// TwinCAT 3 PLC project SODG11_SSCC610_2403701_PLC
// Title: SSCC6.10
// Company: Sodecia GTAC
// Author: GTAC FW Team
// ProjectVersion: 6.10
// Description: 20250506_release
// libraries:
//   Tc2_Drive, * (Beckhoff Automation GmbH)
//   Tc2_EtherCAT, * (Beckhoff Automation GmbH)
//   Tc2_Math, * (Beckhoff Automation GmbH)
//   Tc2_MC2, * (Beckhoff Automation GmbH)
//   Tc2_MC2_Drive, * (Beckhoff Automation GmbH)
//   Tc2_MDP, * (Beckhoff Automation GmbH)
//   Tc2_Standard, * (Beckhoff Automation GmbH)
//   Tc2_System, * (Beckhoff Automation GmbH)
//   Tc2_TcpIp, * (Beckhoff Automation GmbH)
//   Tc2_Utilities, * (Beckhoff Automation GmbH)
//   Tc3_EventLogger, * (Beckhoff Automation GmbH)
//   Tc3_IPCDiag, * (Beckhoff Automation GmbH)
//   Tc3_Module, * (Beckhoff Automation GmbH)
// project tree:
//   Data types/ATI/ udt_ATI_Input_20150203.TcDUT, udt_ATI_Output_20150203.TcDUT
//   Data types/Beckhoff IO udts/ udt_AdsAddr.TcDUT, udt_AdsAddr_AX5805.TcDUT, udt_CU1128_20180507.TcDUT, udt_ECATMaster_InfoData_20121206.TcDUT, udt_ECATMaster_Status.TcDUT, udt_ECATMaster_Status_20141211.TcDUT, udt_ECATSlave_Status.TcDUT, udt_ECATSlave_StatusADS.TcDUT, udt_ECATSlave_StatusEXT.TcDUT, udt_ECATSlave_Status_CU1128.TcDUT, udt_ECATSlave_Status_EP9128.TcDUT, udt_EK1100.TcDUT, udt_EK1110_20150812.TcDUT, udt_EK1122.TcDUT, udt_EL1004.TcDUT, udt_EL1004_v2.TcDUT, udt_EL1008.TcDUT, udt_EL1904.TcDUT, udt_EL1904_v2.TcDUT, udt_EL2008.TcDUT, udt_EL2008_STAT.TcDUT, udt_EL2008_v2.TcDUT, udt_EL2622.TcDUT, udt_EL2622_STAT.TcDUT, udt_EL2904.TcDUT, udt_EL2904RO.TcDUT, udt_EL2904RO_v2.TcDUT, udt_EL3052.TcDUT, udt_EL6692_20121204.TcDUT, udt_EL6695_20151028.TcDUT, udt_EL6731.TcDUT, udt_EL6900_CMD.TcDUT, udt_EL6900_CMD_20121204.TcDUT, udt_EL6900_DeviceInfoData_20160426.TcDUT, udt_EL6900_SafetyGroup_CMD.TcDUT, udt_EL6900_SafetyGroup_STAT.TcDUT, udt_EL6900_STAT.TcDUT, udt_EL6900_STAT_20160426.TcDUT, udt_EL94xx.TcDUT, udt_EP1008_002.TcDUT, udt_EP1008_002_v2.TcDUT, udt_EP1111.TcDUT, udt_EP1908_002.TcDUT, udt_EP1918.TcDUT, udt_EP1918_CMD_20250213.TcDUT, udt_EP1918_STAT_20250213.TcDUT, udt_EP2028_002.TcDUT, udt_EP2028_002_STAT.TcDUT, udt_EP2028_002_v2.TcDUT, udt_EP2328_0002.TcDUT, udt_EP2624.TcDUT, udt_EP2624_STAT.TcDUT, udt_EP3174_0002.TcDUT, udt_EP6224.TcDUT, udt_EP6224_CMD.TcDUT, udt_EP6224_I.TcDUT, udt_EP9128_20250704.TcDUT, udt_EP9214_CH_CMD_20250704.TcDUT, udt_EP9214_CH_STAT_20250704.TcDUT, udt_EP9214_CMD_20250704.TcDUT, udt_EP9214_DEV_CMD_20250704.TcDUT, udt_EP9214_DEV_STAT_20250704.TcDUT, udt_EP9214_STAT_20250704.TcDUT, udt_EP9224_CH_CMD_20161207.TcDUT, udt_EP9224_CH_STAT_20161207.TcDUT, udt_EP9224_CMD_20161207.TcDUT, udt_EP9224_DEV_CMD_20161207.TcDUT, udt_EP9224_DEV_STAT_20161207.TcDUT, udt_EP9224_STAT_20161207.TcDUT, udt_ProfiMaster_Status.TcDUT, udt_ProfiNet_Status.TcDUT, udt_ProfiNode_Status.TcDUT, udt_SMB_Status_20141211.TcDUT
//   Data types/Discrete Image udts/ udt_ATIxx_Image_20151104.TcDUT, udt_Drive_Image_20160804.TcDUT, udt_Drive_Image_20190816.TcDUT, udt_ECATMaster_Image_20220224.TcDUT, udt_ECATNodeConfig_20200729.TcDUT, udt_ECATNodeData_20221507.TcDUT, udt_ECAT_NodeImage_20200618.TcDUT, udt_EOATxx_Image_20170607.TcDUT, udt_EOATxx_Image_20220715.TcDUT, udt_ESWxx_Image_20150814.TcDUT, udt_FixXX_Input_Image_20180202.TcDUT, udt_FixXX_Output_Image_20220715.TcDUT, udt_FixXX_Output_Image_20250721_CUSTOM.TcDUT, udt_FixXX_Persistent_Input.TcDUT, udt_Fronius_Status_20170531.TcDUT, udt_ICxx_Image.TcDUT, udt_ICxx_Image_20201104.TcDUT, udt_MDxx_Image_20251008.TcDUT, udt_NutWeldLVDT_Input_Image_20250616.TcDUT, udt_NutWeldLVDT_Output_Image_20250616.TcDUT, udt_NWx_Image.TcDUT, udt_ISxx_Image_20241121.TcDUT, udt_PEDxx_Image_20170725.TcDUT, udt_PEDxx_Image_20240808.TcDUT, udt_Reamerxx_Image_20180405.TcDUT, udt_RobotDiscreteNode_Image.TcDUT, udt_RobotDiscreteNode_ImageFSOE_20151028.TcDUT, udt_RobotDiscreteNode_ImageSSCCv46wSAFEOP_20131903.TcDUT, udt_RobotDiscreteNode_ImageSSCCv46_20121204.TcDUT, udt_RobotDiscreteNode_ImageSSCCv46_20131001.TcDUT, udt_SDx_Image.TcDUT, udt_SSxx_Image_20150814.TcDUT, udt_SSxx_Image_20250704.TcDUT, udt_STxx_DiscreteNode_20200212.TcDUT, udt_WaterStand_Image_20220131.TcDUT
//   Data types/Emhart udts/ udt_Emhart_DCE1800_Inputold.TcDUT, udt_Emhart_DCE1800_Outputold.TcDUT, udt_Emhart_TE1500_Input.TcDUT, udt_Emhart_TE1500_Inputa.TcDUT, udt_Emhart_TE1500_Output.TcDUT, udt_Emhart_TE1500_Outputa.TcDUT
//   Data types/FSoE udts/ ST_FSoE_02Byte.TcDUT, ST_FSoE_04Byte.TcDUT, ST_FSoE_06Byte.TcDUT, ST_FSoE_08Byte.TcDUT, ST_FSoE_10Byte.TcDUT, ST_FSoE_12Byte.TcDUT, ST_FSoE_14Byte.TcDUT
//   Data types/Generic udts/ udt_Generic_AdsAddr.TcDUT, udt_Generic_EP9214_20250714.TcDUT, udt_Generic_IC_20150928.TcDUT, udt_Generic_Nok_Data_Grid_20251208.TcDUT, udt_Generic_NutWeldLVDTConfig_20250612.TcDUT, udt_Generic_PD_20220906.TcDUT, udt_Generic_Production_20221007.TcDUT, udt_Generic_ProductReportData_20240909.TcDUT, udt_Generic_Robot_20161202.TcDUT, udt_Generic_Robot_20250711_CUSTOM.TcDUT, udt_Generic_Robot_FBIN_CUSTOM.TcDUT, udt_Generic_Robot_FBIN_20250711_CUSTOM.TcDUT, udt_Generic_Robot_Options_20170531.TcDUT, udt_Generic_Sensor_States_20170801.TcDUT, udt_Generic_ServoDrive_FBIN_20211214.TcDUT, udt_Generic_ShiftCommonConfig_20220420.TcDUT, udt_Generic_ShiftConfigTOD_20160527.TcDUT, udt_Generic_ShiftConfigUDINT_20160531.TcDUT, udt_Generic_ShiftConfig_20160519.TcDUT, udt_IVxx_Input_Image_20250812.TcDUT
//   Data types/Graco udts/ udt_Graco_Input.TcDUT, udt_Graco_Outputs.TcDUT
//   Data types/HardwareDiags/ E_State.TcDUT, udt_HardwareDiags.TcDUT
//   Data types/Keyence/ udt_IV2_DiscreteImage.TcDUT, udt_IV2_Inputs.TcDUT, udt_IV2_Outputs.TcDUT
//   Data types/Robot_udts/ udt_EtherCAT_Kuka_InputBits_20121204.TcDUT, udt_EtherCAT_Kuka_OutputBits_20121204.TcDUT, udt_EtherCAT_Motoman_Input_20151105.TcDUT, udt_EtherCAT_Motoman_Output_20151105.TcDUT, udt_GenericRobot_AnyFieldbus_Input58Bytes.TcDUT, udt_GenericRobot_AnyFieldbus_InputBytes_20220421.TcDUT, udt_GenericRobot_AnyFieldbus_Output58Bytes.TcDUT, udt_GenericRobot_AnyFieldbus_OutputBytes_20220421.TcDUT, udt_GenericRobot_CycleTimes_20170304.TcDUT, udt_Profibus_Motoman_Input.TcDUT, udt_Profibus_Motoman_Input_20121204.TcDUT, udt_Profibus_Motoman_Output.TcDUT, udt_Profibus_Motoman_Output_20121204.TcDUT, udt_SingleAxis_MoveData_20160908.TcDUT, udt_SingleAxis_Position_20150119.TcDUT
//   Data types/Schneider udts/ udt_Schneider_VFD_20180808.TcDUT, udt_Schneider_VFD_Image_20180808.TcDUT, udt_Schneider_VFD_Inputs_20190123.TcDUT, udt_Schneider_VFD_Outputs_20190123.TcDUT
//   Data types/Servo Drive udts/AX5000 Diag/ udt_AX5000Diag.TcDUT
//   Data types/Servo Drive udts/ udt_AX5206_20160804.TcDUT, udt_AX5805_20160804.TcDUT, udt_AX5805_DiagData.TcDUT, udt_EL7211_20150115.TcDUT
//   Data types/SIC/ udt_SIC_Profi_Input_20200727.TcDUT, udt_SIC_Profi_Output_20200727.TcDUT
//   Data types/SmartRay/ udt_PLC_Out_To_SmartRay_IN_20260119.TcDUT, udt_Robot_Out_To_SmartRay_IN_20260119.TcDUT, udt_SmartRay_Out_To_PLC_IN_20260119.TcDUT, udt_SmartRay_Out_To_Robot_IN_20260119.TcDUT
//   Data types/SmartRay/UI udt/ udt_SRxx_DiscreteImage.TcDUT, udt_SRxx_Input_Image.TcDUT, udt_SRxx_ToUI_20260122.TcDUT
//   Data types/SMC udts/ udt_SMC_EX260_Stat.TcDUT, udt_SMC_EX260_ValveBank.TcDUT
//   Data types/Trumpf udts/ udt_EtherCat_Trumpf_InputWords_20171002.TcDUT, udt_EtherCat_Trumpf_OutputWords_20171002.TcDUT, udt_TrumpfImage_20171017.TcDUT
//   Data types/UI udts/GTAC Component IO UI udts/ udt_IVxx_ToUI_20250808.TcDUT, udt_LSRxx_ToUI_20220224.TcDUT, udt_ESWxx_ToUI_20220224.TcDUT, udt_ICxx_ToUI_20220224.TcDUT, udt_MDxx_ToUI_20251008.TcDUT, udt_NWxx_ToUI_20220224.TcDUT, udt_ISxx_ToUI_20241121.TcDUT, udt_ProdReportxx_ToUI_20220224.TcDUT, udt_Rxx_ToUI_20220224.TcDUT, udt_SDxx_ToUI_20220224.TcDUT, udt_SLxx_ToUI_20220224.TcDUT, udt_SSxx_ToUI_20250704.TcDUT, udt_STxx_ToUI_20220224.TcDUT, udt_SDxx_FromUI_20220224.TcDUT, udt_VFDxx_ToUI_20250723.TcDUT
//   Data types/UI udts/ udt_UIcommon_InputPers_20250612.TcDUT, udt_UIcommon_Input_20250616.TcDUT, udt_UIcommon_Output_20251008.TcDUT
//   Global Variables/ Global_Persistent_Variables.TcGVL, Global_Variables.TcGVL, Variable_Configuration.TcGVL
//   POUs/ Faults.TcPOU, GTAC_CONFIG.TcPOU, MAIN.TcPOU, Robot_InterLock_Map.TcPOU
//   POUs/FBs/Diagnose/AX5000 Diag/ FB_AxisDiag_20160810.TcPOU
//   POUs/FBs/ FB_ATI_Changer_20151105.TcPOU, FB_Ax5805_GetInfo_20200609.TcPOU, FB_Clamp_Status.TcPOU, FB_Cylinder_Status.TcPOU, FB_Emhart_20200113.TcPOU, FB_ENET_Com20131205.TcPOU, FB_Graco_Seal_20200716.TcPOU, FB_GTAC_Conveyor_20210303.TcPOU, FB_GTAC_EOAT_20170704.TcPOU, FB_GTAC_ESW_20150814.TcPOU, FB_GTAC_EtherCATMaster_20250723.TcPOU, FB_GTAC_ICxx_20181023.TcPOU, FB_GTAC_IV3_20250730.TcPOU, FB_GTAC_Kuka_CUSTOM.TcPOU, FB_GTAC_Load_Seq_20230302.TcPOU, FB_GTAC_NutWeldLVDT_20250612.TcPOU, FB_GTAC_Motoman_20170531.TcPOU, FB_GTAC_ISxx_20241121.TcPOU, FB_GTAC_Ped_20240808.TcPOU, FB_GTAC_ProcessInterlock_20210526.TcPOU, FB_GTAC_QAcheck_20150529.TcPOU, FB_GTAC_Reamer_20180405.TcPOU, FB_GTAC_MDxx_20251008.TcPOU, FB_GTAC_Reamer_20230328.TcPOU, FB_GTAC_RollDoor_20190108.TcPOU, FB_GTAC_ServoSystem_20211214.TcPOU, FB_GTAC_SS_20250407.TcPOU, FB_GTAC_Valve_20170704.TcPOU, FB_GTAC_WaterStand_20220622.TcPOU, FB_Model_Status.TcPOU, FB_Nok_Datagrid.TcPOU, FB_PP_Sensor.TcPOU, FB_Production_Report_20221007.TcPOU, FB_Pulse_Generator.TcPOU, FB_SCHNEIDERVFD_20180808.TcPOU, FB_SIC_MarkProfi_20200727.TcPOU, FB_SmartRay_20260119.TcPOU, FB_SystemDiags20241206.TcPOU, FB_TripleCylinder_20150625.TcPOU, FB_Trumpf_20180125.TcPOU, FB_UDP_PortCreate20140120.TcPOU, FB_VertiGuard_20260310.TcPOU
//   POUs/Fixtures and EOAT/EOAT/ EOAT04.TcPOU
//   POUs/Fixtures and EOAT/Human/ Fix01.TcPOU, Fix02.TcPOU, Fix03.TcPOU, Fix04.TcPOU, Fix05.TcPOU
//   POUs/Fixtures and EOAT/Internal/ Fix101.TcPOU, Fix102.TcPOU, Fix103.TcPOU, Fix104.TcPOU, Fix105.TcPOU
//   POUs/Fixtures and EOAT/Not_Used/ EOAT01.TcPOU, EOAT02.TcPOU, EOAT03.TcPOU, EOAT05.TcPOU, EOAT06.TcPOU, EOAT07.TcPOU, EOAT08.TcPOU, EOAT09.TcPOU, EOAT10.TcPOU, Fix06.TcPOU, Fix07.TcPOU, Fix08.TcPOU, Fix09.TcPOU, Fix10.TcPOU, Fix106.TcPOU, Fix107.TcPOU, Fix108.TcPOU, Fix109.TcPOU, Fix11.TcPOU, Fix110.TcPOU, Fix111.TcPOU, Fix112.TcPOU, Fix12.TcPOU, Fix13.TcPOU, Fix14.TcPOU, Fix15.TcPOU, Fix16.TcPOU
//   POUs/FUNs/ FUN_GTAC_ASCIItoSTRING.TcPOU, FUN_GTAC_BOOLStoINT.TcPOU, FUN_GTAC_BYTEStoINT.TcPOU, FUN_GTAC_DEGtoINDEX.TcPOU, FUN_GTAC_DINTtoINT.TcPOU, FUN_GTAC_EcatSlaveConnState.TcPOU, FUN_GTAC_EcatSlaveConnState_64bit.TcPOU, FUN_GTAC_FindStringInArray.TcPOU, FUN_GTAC_GenericRobotInputImage_From_KUKAKRC4.TcPOU, FUN_GTAC_GenericRobotInputImage_TO_KUKAKRC4.TcPOU, FUN_GTAC_GenericRobotInputImage_TO_MOTOMAN32.TcPOU, FUN_GTAC_GetNodeFromName.TcPOU, FUN_GTAC_KUKAKRC4_To_GenericRobotOutputImage.TcPOU, FUN_GTAC_MOTOMAN32_TO_GenericRobotOutputImage.TcPOU, FUN_GTAC_NC_Error_Messages.TcPOU, FUN_GTAC_OTSTRUCTtoTOD.TcPOU, FUN_GTAC_OTSTRUCTWrapper.TcPOU, FUN_GTAC_ReturnGrossShiftDuration.TcPOU, FUN_GTAC_ReturnNetShiftDuration.TcPOU, FUN_GTAC_ReturnSetLengthSTR.TcPOU, FUN_GTAC_Scaling.TcPOU, FUN_GTAC_TIMESTRUCTtoTOD.TcPOU, FUN_GTAC_TODtoOTSTRUCT.TcPOU, FUN_GTAC_TODtoUDINT.TcPOU, FUN_GTAC_ZeroSecsInUDINT_Time.TcPOU, FUN_RailMove_To_ICxx.TcPOU
//   POUs/Misc/ Ancillary_Equipment.TcPOU, Cell_Services_Prog.TcPOU, Ped_Stations.TcPOU, Servo_Motion.TcPOU, Task_ID_Record.TcPOU
//   / Standard.TcTTO
// real-time tasks:
//   TASK Standard: cycle T#20ms, priority 11, ADS port 350
// I/O:
//   DEVICE EtherCAT Master (EtherCAT), AmsNetId 172.16.1.120.2.1
//     IC01.T01 (EK1100) [EK1100 EtherCAT Coupler (2A E-Bus)]
//       IC01.T02 (EL6900) [EL6900, TwinSAFE PLC]
//       IC01.T03 (EL1904) [EL1904, 4 Ch. Safety Input 24V, TwinSAFE]
//         modules: Module 1 (FSOES)
//       IC01.T04 (EL1904) [EL1904, 4 Ch. Safety Input 24V, TwinSAFE]
//         modules: Module 1 (FSOES)
//       IC01.T05 (EL1904) [EL1904, 4 Ch. Safety Input 24V, TwinSAFE]
//         modules: Module 1 (FSOES)
//       IC01.T06 (EL1904) [EL1904, 4 Ch. Safety Input 24V, TwinSAFE]
//         modules: Module 1 (FSOES)
//       IC01.T07 (EL1904) [EL1904, 4 Ch. Safety Input 24V, TwinSAFE]
//         modules: Module 1 (FSOES)
//       IC01.T08 (EL1904) [EL1904, 4 Ch. Safety Input 24V, TwinSAFE]
//         modules: Module 1 (FSOES)
//       IC01.T09 (EL2904) [EL2904, 4 Ch. Safety Output 24V, 0.5A, TwinSAFE]
//         modules: Module 1 (FSOES), Module 2 (DO)
//       IC01.T10 (EL2904) [EL2904, 4 Ch. Safety Output 24V, 0.5A, TwinSAFE]
//         modules: Module 1 (FSOES), Module 2 (DO)
//       IC01.T11 (EL9410) [EL9410 E-Bus Power Supplier  (Diagnostics)]
//       IC01.T12 (EL1004) [EL1004 4Ch. Dig. Input 24V, 3ms]
//       IC01.T13 (EL1004) [EL1004 4Ch. Dig. Input 24V, 3ms]
//       IC01.T14 (EL2008) [EL2008 8Ch. Dig. Output 24V, 0.5A]
//       IC01.T15 (EL2622) [EL2622 2Ch. Relay Output, NO (230V AC / 30V DC)]
//       IC01.T16 (EK1122) [EK1122 2 port EtherCAT junction]
//         Fix01.N90 (EP9214-0023) [EP9214-0023 4Ch/4Ch Power Distribution for EtherCAT Box Modules]
//         Fix01.N98  (EP2328-0002) [EP2328-0002 4 CH. Dig. In, 3ms, 4 Ch. Dig. Out 24V, 2A, M12]
//         Fix01.N01 (EP1008-0002) [EP1008-0002 8 Ch. Dig. Input 24V, 3ms, M12]
//         Fix01.N02 (EP1008-0002) [EP1008-0002 8 Ch. Dig. Input 24V, 3ms, M12]
//         Fix01.N03 (EP1008-0002) [EP1008-0002 8 Ch. Dig. Input 24V, 3ms, M12]
//         Fix01.N04 (EP1008-0002) [EP1008-0002 8 Ch. Dig. Input 24V, 3ms, M12]
//         Fix01.N05 (EP1008-0002) [EP1008-0002 8 Ch. Dig. Input 24V, 3ms, M12]
//         Fix01.N06 (EP1008-0002) [EP1008-0002 8 Ch. Dig. Input 24V, 3ms, M12]
//         Fix01.N07 (EP1008-0002) [EP1008-0002 8 Ch. Dig. Input 24V, 3ms, M12]
//         Fix01.N08 (EP1008-0002) [EP1008-0002 8 Ch. Dig. Input 24V, 3ms, M12]
//         Fix01.N09 (EP1008-0002) [EP1008-0002 8 Ch. Dig. Input 24V, 3ms, M12]
//         Fix01.N10 (EP1008-0002) [EP1008-0002 8 Ch. Dig. Input 24V, 3ms, M12]
//         Fix01.N11 (EP1008-0002) [EP1008-0002 8 Ch. Dig. Input 24V, 3ms, M12]
//         Fix01.N12 (EP1008-0002) [EP1008-0002 8 Ch. Dig. Input 24V, 3ms, M12]
//         Fix01.N13 (EP1008-0002) [EP1008-0002 8 Ch. Dig. Input 24V, 3ms, M12]
//         Fix01.N14 (EP1008-0002) [EP1008-0002 8 Ch. Dig. Input 24V, 3ms, M12]
//         Fix01.N15 (EP1008-0002) [EP1008-0002 8 Ch. Dig. Input 24V, 3ms, M12]
//         Fix01.N16 (EP1008-0002) [EP1008-0002 8 Ch. Dig. Input 24V, 3ms, M12]
//         Fix01.N17 (EP1008-0002) [EP1008-0002 8 Ch. Dig. Input 24V, 3ms, M12]
//         Fix01.N18 (EP1008-0002) [EP1008-0002 8 Ch. Dig. Input 24V, 3ms, M12]
//         Fix01.N19 (EP1008-0002) [EP1008-0002 8 Ch. Dig. Input 24V, 3ms, M12]
//         Fix01.N20 (EP1008-0002) [EP1008-0002 8 Ch. Dig. Input 24V, 3ms, M12]
//         Fix01.N21 (EP1008-0002) [EP1008-0002 8 Ch. Dig. Input 24V, 3ms, M12]
//         Fix01.N22 (EP1008-0002) [EP1008-0002 8 Ch. Dig. Input 24V, 3ms, M12]
//         Fix01.N23 (EP1008-0002) [EP1008-0002 8 Ch. Dig. Input 24V, 3ms, M12]
//         Fix01.N24 (EP1008-0002) [EP1008-0002 8 Ch. Dig. Input 24V, 3ms, M12]
//         Fix01.N25 (EP1008-0002) [EP1008-0002 8 Ch. Dig. Input 24V, 3ms, M12]
//         Fix01.N26 (EP1008-0002) [EP1008-0002 8 Ch. Dig. Input 24V, 3ms, M12]
//         Fix01.N27 (EP1008-0002) [EP1008-0002 8 Ch. Dig. Input 24V, 3ms, M12]
//         Fix01.N28 (EP1008-0002) [EP1008-0002 8 Ch. Dig. Input 24V, 3ms, M12]
//         Fix01.N29 (EP1008-0002) [EP1008-0002 8 Ch. Dig. Input 24V, 3ms, M12]
//         Fix01.N30 (EP1008-0002) [EP1008-0002 8 Ch. Dig. Input 24V, 3ms, M12] (disabled)
//         Fix01.N31 (EP1008-0002) [EP1008-0002 8 Ch. Dig. Input 24V, 3ms, M12] (disabled)
//         Fix01.N100 (EX260-SEC1) [EX260-SEC1 EtherCAT SI Unit (32DO_PNP) Rev1.2]
//         Fix01.N101 (EX260-SEC1) [EX260-SEC1 EtherCAT SI Unit (32DO_PNP) Rev1.2]
//         Fix02.N90 (EP9214-0023) [EP9214-0023 4Ch/4Ch Power Distribution for EtherCAT Box Modules]
//         Fix02.N98(EP2328-0002) [EP2328-0002 4 CH. Dig. In, 3ms, 4 Ch. Dig. Out 24V, 2A, M12]
//         Fix02.N01 (EP1008-0002) [EP1008-0002 8 Ch. Dig. Input 24V, 3ms, M12]
//         Fix02.N02 (EP1008-0002) [EP1008-0002 8 Ch. Dig. Input 24V, 3ms, M12]
//         Fix02.N03 (EP1008-0002) [EP1008-0002 8 Ch. Dig. Input 24V, 3ms, M12]
//         Fix02.N04 (EP1008-0002) [EP1008-0002 8 Ch. Dig. Input 24V, 3ms, M12]
//         Fix02.N05 (EP1008-0002) [EP1008-0002 8 Ch. Dig. Input 24V, 3ms, M12]
//         Fix02.N06 (EP1008-0002) [EP1008-0002 8 Ch. Dig. Input 24V, 3ms, M12]
//         Fix02.N07 (EP1008-0002) [EP1008-0002 8 Ch. Dig. Input 24V, 3ms, M12]
//         Fix02.N08 (EP1008-0002) [EP1008-0002 8 Ch. Dig. Input 24V, 3ms, M12]
//         Fix02.N09 (EP1008-0002) [EP1008-0002 8 Ch. Dig. Input 24V, 3ms, M12]
//         Fix02.N10 (EP1008-0002) [EP1008-0002 8 Ch. Dig. Input 24V, 3ms, M12]
//         Fix02.N11 (EP1008-0002) [EP1008-0002 8 Ch. Dig. Input 24V, 3ms, M12]
//         Fix02.N12 (EP1008-0002) [EP1008-0002 8 Ch. Dig. Input 24V, 3ms, M12]
//         Fix02.N13 (EP1008-0002) [EP1008-0002 8 Ch. Dig. Input 24V, 3ms, M12]
//         Fix02.N14 (EP1008-0002) [EP1008-0002 8 Ch. Dig. Input 24V, 3ms, M12]
//         Fix02.N15 (EP1008-0002) [EP1008-0002 8 Ch. Dig. Input 24V, 3ms, M12]
//         Fix02.N16 (EP1008-0002) [EP1008-0002 8 Ch. Dig. Input 24V, 3ms, M12]
//         Fix02.N17 (EP1008-0002) [EP1008-0002 8 Ch. Dig. Input 24V, 3ms, M12]
//         Fix02.N18 (EP1008-0002) [EP1008-0002 8 Ch. Dig. Input 24V, 3ms, M12]
//         Fix02.N19 (EP1008-0002) [EP1008-0002 8 Ch. Dig. Input 24V, 3ms, M12]
//         Fix02.N20 (EP1008-0002) [EP1008-0002 8 Ch. Dig. Input 24V, 3ms, M12]
//         Fix02.N21 (EP1008-0002) [EP1008-0002 8 Ch. Dig. Input 24V, 3ms, M12]
//         Fix02.N22 (EP1008-0002) [EP1008-0002 8 Ch. Dig. Input 24V, 3ms, M12]
//         Fix02.N23 (EP1008-0002) [EP1008-0002 8 Ch. Dig. Input 24V, 3ms, M12]
//         Fix02.N24 (EP1008-0002) [EP1008-0002 8 Ch. Dig. Input 24V, 3ms, M12]
//         Fix02.N25 (EP1008-0002) [EP1008-0002 8 Ch. Dig. Input 24V, 3ms, M12]
//         Fix02.N26 (EP1008-0002) [EP1008-0002 8 Ch. Dig. Input 24V, 3ms, M12]
//         Fix02.N27 (EP1008-0002) [EP1008-0002 8 Ch. Dig. Input 24V, 3ms, M12]
//         Fix02.N28(EP1008-0002) [EP1008-0002 8 Ch. Dig. Input 24V, 3ms, M12]
//         Fix02.N29 (EP1008-0002) [EP1008-0002 8 Ch. Dig. Input 24V, 3ms, M12]
//         Fix02.N30 (EP1008-0002) [EP1008-0002 8 Ch. Dig. Input 24V, 3ms, M12] (disabled)
//         Fix02.N31 (EP1008-0002) [EP1008-0002 8 Ch. Dig. Input 24V, 3ms, M12] (disabled)
//         Fix02.N100 (EX260-SEC1) [EX260-SEC1 EtherCAT SI Unit (32DO_PNP) Rev1.2]
//         Fix02.N101 (EX260-SEC1) [EX260-SEC1 EtherCAT SI Unit (32DO_PNP) Rev1.2]
//       IC01.T17 (EL9011) [EL9011 End Terminal]
//     MD01.N01 (EP1918-0002) [EP1918, 8Ch. Safety Input 24V, TwinSAFE]
//       modules: Module 2 (FSLOGIC)
//     MD01.N02 (EP1008-0002) [EP1008-0002 8 Ch. Dig. Input 24V, 3ms, M12]
//     MD01.N03 (EP2624-0002) [EP2624-0002 4Ch. Relay Output, NO (125V AC / 30V DC)]
//     MD02.N01 (EP1918-0002) [EP1918, 8Ch. Safety Input 24V, TwinSAFE]
//       modules: Module 2 (FSLOGIC)
//     MD02.N02 (EP1008-0002) [EP1008-0002 8 Ch. Dig. Input 24V, 3ms, M12]
//     MD02.N03 (EP2624-0002) [EP2624-0002 4Ch. Relay Output, NO (125V AC / 30V DC)]
//     IC02.T01 (EK1100) [EK1100 EtherCAT Coupler (2A E-Bus)]
//       IC02.T02 (EL6900) [EL6900, TwinSAFE PLC]
//       IC02.T03 (EL1904) [EL1904, 4 Ch. Safety Input 24V, TwinSAFE]
//         modules: Module 1 (FSOES)
//       IC02.T04 (EL1904) [EL1904, 4 Ch. Safety Input 24V, TwinSAFE]
//         modules: Module 1 (FSOES)
//       IC02.T05 (EL1904) [EL1904, 4 Ch. Safety Input 24V, TwinSAFE]
//         modules: Module 1 (FSOES)
//       IC02.T06 (EL1904) [EL1904, 4 Ch. Safety Input 24V, TwinSAFE]
//         modules: Module 1 (FSOES)
//       IC02.T07 (EL1904) [EL1904, 4 Ch. Safety Input 24V, TwinSAFE]
//         modules: Module 1 (FSOES)
//       IC02.T08 (EL1904) [EL1904, 4 Ch. Safety Input 24V, TwinSAFE]
//         modules: Module 1 (FSOES)
//       IC02.T09 (EL2904) [EL2904, 4 Ch. Safety Output 24V, 0.5A, TwinSAFE]
//         modules: Module 1 (FSOES), Module 2 (DO)
//       IC02.T10 (EL2904) [EL2904, 4 Ch. Safety Output 24V, 0.5A, TwinSAFE]
//         modules: Module 1 (FSOES), Module 2 (DO)
//       IC02.T11 (EL9410) [EL9410 E-Bus Power Supplier  (Diagnostics)]
//       IC02.T12 (EL1004) [EL1004 4Ch. Dig. Input 24V, 3ms]
//       IC02.T13 (EL1004) [EL1004 4Ch. Dig. Input 24V, 3ms]
//       IC02.T14 (EL2008) [EL2008 8Ch. Dig. Output 24V, 0.5A]
//       IC02.T15 (EL2622) [EL2622 2Ch. Relay Output, NO (230V AC / 30V DC)]
//       IC02.T16 (EK1122) [EK1122 2 port EtherCAT junction]
//         Fix03.N90 (EP9214-0023) [EP9214-0023 4Ch/4Ch Power Distribution for EtherCAT Box Modules]
//         Fix03.N98  (EP2328-0002) [EP2328-0002 4 CH. Dig. In, 3ms, 4 Ch. Dig. Out 24V, 2A, M12]
//         Fix03.N01 (EP1008-0002) [EP1008-0002 8 Ch. Dig. Input 24V, 3ms, M12]
//         Fix03.N02 (EP1008-0002) [EP1008-0002 8 Ch. Dig. Input 24V, 3ms, M12]
//         Fix03.N03 (EP1008-0002) [EP1008-0002 8 Ch. Dig. Input 24V, 3ms, M12]
//         Fix03.N04 (EP1008-0002) [EP1008-0002 8 Ch. Dig. Input 24V, 3ms, M12]
//         Fix03.N05 (EP1008-0002) [EP1008-0002 8 Ch. Dig. Input 24V, 3ms, M12]
//         Fix03.N06 (EP1008-0002) [EP1008-0002 8 Ch. Dig. Input 24V, 3ms, M12]
//         Fix03.N07 (EP1008-0002) [EP1008-0002 8 Ch. Dig. Input 24V, 3ms, M12]
//         Fix03.N08 (EP1008-0002) [EP1008-0002 8 Ch. Dig. Input 24V, 3ms, M12]
//         Fix03.N09 (EP1008-0002) [EP1008-0002 8 Ch. Dig. Input 24V, 3ms, M12]
//         Fix03.N10 (EP1008-0002) [EP1008-0002 8 Ch. Dig. Input 24V, 3ms, M12]
//         Fix03.N11 (EP1008-0002) [EP1008-0002 8 Ch. Dig. Input 24V, 3ms, M12]
//         Fix03.N12 (EP1008-0002) [EP1008-0002 8 Ch. Dig. Input 24V, 3ms, M12]
//         Fix03.N13 (EP1008-0002) [EP1008-0002 8 Ch. Dig. Input 24V, 3ms, M12]
//         Fix03.N14 (EP1008-0002) [EP1008-0002 8 Ch. Dig. Input 24V, 3ms, M12]
//         Fix03.N15 (EP1008-0002) [EP1008-0002 8 Ch. Dig. Input 24V, 3ms, M12]
//         Fix03.N16 (EP1008-0002) [EP1008-0002 8 Ch. Dig. Input 24V, 3ms, M12]
//         Fix03.N17 (EP1008-0002) [EP1008-0002 8 Ch. Dig. Input 24V, 3ms, M12]
//         Fix03.N18 (EP1008-0002) [EP1008-0002 8 Ch. Dig. Input 24V, 3ms, M12]
//         Fix03.N19 (EP1008-0002) [EP1008-0002 8 Ch. Dig. Input 24V, 3ms, M12]
//         Fix03.N20 (EP1008-0002) [EP1008-0002 8 Ch. Dig. Input 24V, 3ms, M12]
//         Fix03.N21 (EP1008-0002) [EP1008-0002 8 Ch. Dig. Input 24V, 3ms, M12]
//         Fix03.N22 (EP1008-0002) [EP1008-0002 8 Ch. Dig. Input 24V, 3ms, M12]
//         Fix03.N100 (EX260-SEC1) [EX260-SEC1 EtherCAT SI Unit (32DO_PNP) Rev1.2]
//         Fix04.N90 (EP9214-0023) [EP9214-0023 4Ch/4Ch Power Distribution for EtherCAT Box Modules]
//         Fix04.N98  (EP2328-0002) [EP2328-0002 4 CH. Dig. In, 3ms, 4 Ch. Dig. Out 24V, 2A, M12]
//         Fix04.N01 (EP1008-0002) [EP1008-0002 8 Ch. Dig. Input 24V, 3ms, M12]
//         Fix04.N02 (EP1008-0002) [EP1008-0002 8 Ch. Dig. Input 24V, 3ms, M12]
//         Fix04.N03 (EP1008-0002) [EP1008-0002 8 Ch. Dig. Input 24V, 3ms, M12]
//         Fix04.N04 (EP1008-0002) [EP1008-0002 8 Ch. Dig. Input 24V, 3ms, M12]
//         Fix04.N05 (EP1008-0002) [EP1008-0002 8 Ch. Dig. Input 24V, 3ms, M12]
//         Fix04.N06 (EP1008-0002) [EP1008-0002 8 Ch. Dig. Input 24V, 3ms, M12]
//         Fix04.N07 (EP1008-0002) [EP1008-0002 8 Ch. Dig. Input 24V, 3ms, M12]
//         Fix04.N08 (EP1008-0002) [EP1008-0002 8 Ch. Dig. Input 24V, 3ms, M12]
//         Fix04.N09 (EP1008-0002) [EP1008-0002 8 Ch. Dig. Input 24V, 3ms, M12]
//         Fix04.N10 (EP1008-0002) [EP1008-0002 8 Ch. Dig. Input 24V, 3ms, M12]
//         Fix04.N11 (EP1008-0002) [EP1008-0002 8 Ch. Dig. Input 24V, 3ms, M12]
//         Fix04.N12 (EP1008-0002) [EP1008-0002 8 Ch. Dig. Input 24V, 3ms, M12]
//         Fix04.N13 (EP1008-0002) [EP1008-0002 8 Ch. Dig. Input 24V, 3ms, M12]
//         Fix04.N14 (EP1008-0002) [EP1008-0002 8 Ch. Dig. Input 24V, 3ms, M12]
//         Fix04.N15 (EP1008-0002) [EP1008-0002 8 Ch. Dig. Input 24V, 3ms, M12]
//         Fix04.N16 (EP1008-0002) [EP1008-0002 8 Ch. Dig. Input 24V, 3ms, M12]
//         Fix04.N17 (EP1008-0002) [EP1008-0002 8 Ch. Dig. Input 24V, 3ms, M12]
//         Fix04.N18 (EP1008-0002) [EP1008-0002 8 Ch. Dig. Input 24V, 3ms, M12]
//         Fix04.N19 (EP1008-0002) [EP1008-0002 8 Ch. Dig. Input 24V, 3ms, M12]
//         Fix04.N20 (EP1008-0002) [EP1008-0002 8 Ch. Dig. Input 24V, 3ms, M12]
//         Fix04.N21 (EP1008-0002) [EP1008-0002 8 Ch. Dig. Input 24V, 3ms, M12]
//         Fix04.N22 (EP1008-0002) [EP1008-0002 8 Ch. Dig. Input 24V, 3ms, M12] (disabled)
//         Fix04.N100 (EX260-SEC1) [EX260-SEC1 EtherCAT SI Unit (32DO_PNP) Rev1.2]
//       IC02.T17 (EL9011) [EL9011 End Terminal]
//     ESW03.N01 (EP1908) [EP1908, 8 Ch. Safety Input 24V, TwinSAFE]
//       modules: Module 1 (FSOE)
//     R5.T01 (EK1100) [EK1100 EtherCAT Coupler (2A E-Bus)]
//       R5.T02 (EL6900) [EL6900, TwinSAFE PLC]
//       R5.T03 (EL1904) [EL1904, 4 Ch. Safety Input 24V, TwinSAFE]
//         modules: Module 1 (FSOES)
//       R5.T04 (EK1122) [EK1122 2 port EtherCAT junction]
//         R5.Reamer[1].N01 (EP1008-0002) [EP1008-0002 8 Ch. Dig. Input 24V, 3ms, M12]
//         R5.Reamer[1].N30 (EP2028-0002) [EP2028-0002 8 Ch. Dig. Output 24V, 2A, M12]
//     R5.RT02 (EL6695-1001) [KRC4 secondary EL6695-1001]
//       modules: Module 1 (Sync Inputs), Module 2 (Safety Data (8 Byte)), Module 3 (Default IO)
//     R6.T01 (EK1100) [EK1100 EtherCAT Coupler (2A E-Bus)]
//       R6.T02 (EL6900) [EL6900, TwinSAFE PLC]
//       R6.T03 (EL1904) [EL1904, 4 Ch. Safety Input 24V, TwinSAFE]
//         modules: Module 1 (FSOES)
//       R6.T04 (EK1122) [EK1122 2 port EtherCAT junction]
//         R6.Reamer[1].N01 (EP1008-0002) [EP1008-0002 8 Ch. Dig. Input 24V, 3ms, M12]
//         R6.Reamer[1].N30 (EP2028-0002) [EP2028-0002 8 Ch. Dig. Output 24V, 2A, M12]
//     R6.RT02 (EL6695-1001) [KRC4 secondary EL6695-1001]
//       modules: Module 1 (Sync Inputs), Module 2 (Safety Data (8 Byte)), Module 3 (Default IO)
//     R10.T01 (EK1100) [EK1100 EtherCAT Coupler (2A E-Bus)]
//       R10.T02 (EL6900) [EL6900, TwinSAFE PLC]
//       R10.T03 (EL1904) [EL1904, 4 Ch. Safety Input 24V, TwinSAFE]
//         modules: Module 1 (FSOES)
//       R10.T04 (EK1122) [EK1122 2 port EtherCAT junction]
//     R10.RT02 (EL6695-1001) [KRC4 secondary EL6695-1001]
//       modules: Module 1 (Sync Inputs), Module 2 (Safety Data (8 Byte)), Module 3 (Default IO)
//     R11.T01 (EK1100) [EK1100 EtherCAT Coupler (2A E-Bus)]
//       R11.T02 (EL6900) [EL6900, TwinSAFE PLC]
//       R11.T03 (EL1904) [EL1904, 4 Ch. Safety Input 24V, TwinSAFE]
//         modules: Module 1 (FSOES)
//       R11.T04 (EK1122) [EK1122 2 port EtherCAT junction]
//     R11.RT02 (EL6695-1001) [KRC4 secondary EL6695-1001]
//       modules: Module 1 (Sync Inputs), Module 2 (Safety Data (8 Byte)), Module 3 (Default IO)
//     IC03.T01 (EK1100) [EK1100 EtherCAT Coupler (2A E-Bus)]
//       IC03.T02 (EL6900) [EL6900, TwinSAFE PLC]
//       IC03.T03 (EL1904) [EL1904, 4 Ch. Safety Input 24V, TwinSAFE]
//         modules: Module 1 (FSOES)
//       IC03.T04 (EL1904) [EL1904, 4 Ch. Safety Input 24V, TwinSAFE]
//         modules: Module 1 (FSOES)
//       IC03.T05 (EL1904) [EL1904, 4 Ch. Safety Input 24V, TwinSAFE]
//         modules: Module 1 (FSOES)
//       IC03.T06 (EL1904) [EL1904, 4 Ch. Safety Input 24V, TwinSAFE]
//         modules: Module 1 (FSOES)
//       IC03.T07 (EL1904) [EL1904, 4 Ch. Safety Input 24V, TwinSAFE]
//         modules: Module 1 (FSOES)
//       IC03.T08 (EL1904) [EL1904, 4 Ch. Safety Input 24V, TwinSAFE]
//         modules: Module 1 (FSOES)
//       IC03.T09 (EL2904) [EL2904, 4 Ch. Safety Output 24V, 0.5A, TwinSAFE]
//         modules: Module 1 (FSOES), Module 2 (DO)
//       IC03.T10 (EL2904) [EL2904, 4 Ch. Safety Output 24V, 0.5A, TwinSAFE]
//         modules: Module 1 (FSOES), Module 2 (DO)
//       IC03.T11 (EL9410) [EL9410 E-Bus Power Supplier  (Diagnostics)]
//       IC03.T12 (EL1004) [EL1004 4Ch. Dig. Input 24V, 3ms]
//       IC03.T13 (EL1004) [EL1004 4Ch. Dig. Input 24V, 3ms]
//       IC03.T14 (EL2008) [EL2008 8Ch. Dig. Output 24V, 0.5A]
//       IC03.T15 (EL2622) [EL2622 2Ch. Relay Output, NO (230V AC / 30V DC)]
//       IC03.T16 (EK1122) [EK1122 2 port EtherCAT junction]
//         Fix05.N01 (EP1008-0002) [EP1008-0002 8 Ch. Dig. Input 24V, 3ms, M12]
//         Fix05.N02 (EP1008-0002) [EP1008-0002 8 Ch. Dig. Input 24V, 3ms, M12]
//         Fix05.N03 (EP1008-0002) [EP1008-0002 8 Ch. Dig. Input 24V, 3ms, M12]
//         Fix05.N04 (EP1008-0002) [EP1008-0002 8 Ch. Dig. Input 24V, 3ms, M12]
//         Fix05.N100 (EX260-SEC1) [EX260-SEC1 EtherCAT SI Unit (32DO_PNP) Rev1.2]
//         Fix102.N01 (EP1008-0002) [EP1008-0002 8 Ch. Dig. Input 24V, 3ms, M12]
//         Fix102.N02 (EP1008-0002) [EP1008-0002 8 Ch. Dig. Input 24V, 3ms, M12]
//         Fix102.N03 (EP1008-0002) [EP1008-0002 8 Ch. Dig. Input 24V, 3ms, M12]
//         Fix102.N04 (EP1008-0002) [EP1008-0002 8 Ch. Dig. Input 24V, 3ms, M12]
//         Fix102.N100 (EX260-SEC1) [EX260-SEC1 EtherCAT SI Unit (32DO_PNP) Rev1.2]
//         QA_Fix102CAM1 (DL-EC1A) [DL-EC1A] (disabled)
//         QA_Fix102CAM2 (DL-EC1A)
//       IC03.T17 (EL9011) [EL9011 End Terminal]
//     ESW02.N01 (EP1908) [EP1908, 8 Ch. Safety Input 24V, TwinSAFE]
//       modules: Module 1 (FSOE)
//     IS01.T01 (EK1100) [EK1100 EtherCAT Coupler (2A E-Bus)]
//       IS01.T02 (EL6900) [EL6900, TwinSAFE PLC]
//       IS01.T03 (EL1904) [EL1904, 4 Ch. Safety Input 24V, TwinSAFE]
//         modules: Module 1 (FSOES)
//       IS01.T04 (EL2904) [EL2904, 4 Ch. Safety Output 24V, 0.5A, TwinSAFE]
//         modules: Module 1 (FSOES), Module 2 (DO)
//       IS01.T05 (EL6731) [EL6731 PROFIBUS DP Master]
//       IS01.T06 (EK1110) [EK1110 EtherCAT extension]
//     SS01.N01 (EP9128-0021) [EP9128-0021 8x EtherCAT junction]
//       Fix101.N01 (EP1008-0002) [EP1008-0002 8 Ch. Dig. Input 24V, 3ms, M12]
//       Fix101.N02 (EP1008-0002) [EP1008-0002 8 Ch. Dig. Input 24V, 3ms, M12]
//       Fix101.N03 (EP1008-0002) [EP1008-0002 8 Ch. Dig. Input 24V, 3ms, M12]
//       Fix101.N04 (EP1008-0002) [EP1008-0002 8 Ch. Dig. Input 24V, 3ms, M12]
//       Fix101.N100 (EX260-SEC1) [EX260-SEC1 EtherCAT SI Unit (32DO_PNP) Rev1.2]
//       VertiGuard.N01 (EP2028-0002) [EP2028-0002 8 Ch. Dig. Output 24V, 2A, M12]
//       VertiGuard.N02 (EP1908) [EP1908, 8 Ch. Safety Input 24V, TwinSAFE ]
//         modules: Module 1 (FSOE)
//       Term 299 (EP9128-1021) [EP9128-1021 8x EtherCAT junction - Dev A]
//         Fix103.N01 (EP1008-0002) [EP1008-0002 8 Ch. Dig. Input 24V, 3ms, M12] (disabled)
//         Fix103.N02 (EP1008-0002) [EP1008-0002 8 Ch. Dig. Input 24V, 3ms, M12] (disabled)
//         VFD01 (ATV320 EtherCAT) [ATV320 EtherCAT] (disabled)
//         Fix104.N01 (EP1008-0002) [EP1008-0002 8 Ch. Dig. Input 24V, 3ms, M12] (disabled)
//         Fix104.N02 (EP1008-0002) [EP1008-0002 8 Ch. Dig. Input 24V, 3ms, M12] (disabled)
//         VFD02 (ATV320 EtherCAT) [ATV320 EtherCAT] (disabled)
//         Fix105.N01 (EP1008-0002)
//         Fix105.N02 (EP1008-0002)
//       Term 301 (EP9128-2021) [EP9128-2021 8x EtherCAT junction - Dev B]
//     SS01.N02 (EP1008-0002) [EP1008-0002 8 Ch. Dig. Input 24V, 3ms, M12]
//     SS01.N03 (EP2028-0002) [EP2028-0002 8 Ch. Dig. Output 24V, 2A, M12]
//     SS01.N04 (EP9214-0023) [EP9214-0023 4Ch/4Ch Power Distribution for EtherCAT Box Modules]
//     R4.T01 (EK1100) [EK1100 EtherCAT Coupler (2A E-Bus)]
//       R4.T02 (EL6900) [EL6900, TwinSAFE PLC]
//       R4.T03 (EL1904) [EL1904, 4 Ch. Safety Input 24V, TwinSAFE]
//         modules: Module 1 (FSOES)
//       R4.T04 (EK1122) [EK1122 2 port EtherCAT junction]
//         EOAT04.N00 (EP1111-0002) [EP1111-0000 ID-Switch]
//         EOAT04.N01 (EP1008-0002) [EP1008-0002 8 Ch. Dig. Input 24V, 3ms, M12]
//         EOAT04.N02 (EP1008-0002) [EP1008-0002 8 Ch. Dig. Input 24V, 3ms, M12]
//         EOAT04.N03 (EP1008-0002) [EP1008-0002 8 Ch. Dig. Input 24V, 3ms, M12]
//         EOAT04.N04 (EP1008-0002) [EP1008-0002 8 Ch. Dig. Input 24V, 3ms, M12]
//         EOAT04.N100 (EX260-SEC1) [EX260-SEC1 EtherCAT SI Unit (32DO_PNP) Rev1.2]
//     R4.RT02 (EL6695-1001) [KRC4 secondary EL6695-1001]
//       modules: Module 1 (Sync Inputs), Module 2 (Safety Data (8 Byte)), Module 3 (Default IO)
//     R1.T01 (EK1100) [EK1100 EtherCAT Coupler (2A E-Bus)]
//       R1.T02 (EL6900) [EL6900, TwinSAFE PLC]
//       R1.T03 (EL1904) [EL1904, 4 Ch. Safety Input 24V, TwinSAFE]
//         modules: Module 1 (FSOES)
//       R1.T04 (EK1122) [EK1122 2 port EtherCAT junction]
//         R1.Reamer[1].N01 (EP1008-0002) [EP1008-0002 8 Ch. Dig. Input 24V, 3ms, M12]
//         R1.Reamer[1].N30 (EP2028-0002) [EP2028-0002 8 Ch. Dig. Output 24V, 2A, M12]
//     R1.RT02 (EL6695-1001) [KRC4 secondary EL6695-1001]
//       modules: Module 1 (Sync Inputs), Module 2 (Safety Data (8 Byte)), Module 3 (Default IO)
//     R2.T01 (EK1100) [EK1100 EtherCAT Coupler (2A E-Bus)]
//       R2.T02 (EL6900) [EL6900, TwinSAFE PLC]
//       R2.T03 (EL1904) [EL1904, 4 Ch. Safety Input 24V, TwinSAFE]
//         modules: Module 1 (FSOES)
//       R2.T04 (EK1122) [EK1122 2 port EtherCAT junction]
//         R2.Reamer[1].N01 (EP1008-0002) [EP1008-0002 8 Ch. Dig. Input 24V, 3ms, M12]
//         R2.Reamer[1].N30 (EP2028-0002) [EP2028-0002 8 Ch. Dig. Output 24V, 2A, M12]
//     R2.RT02 (EL6695-1001) [KRC4 secondary EL6695-1001]
//       modules: Module 1 (Sync Inputs), Module 2 (Safety Data (8 Byte)), Module 3 (Default IO)
//     R3.T01 (EK1100) [EK1100 EtherCAT Coupler (2A E-Bus)]
//       R3.T02 (EL6900) [EL6900, TwinSAFE PLC]
//       R3.T03 (EL1904) [EL1904, 4 Ch. Safety Input 24V, TwinSAFE]
//         modules: Module 1 (FSOES)
//       R3.T04 (EK1122) [EK1122 2 port EtherCAT junction]
//         R3.Reamer[1].N01 (EP1008-0002) [EP1008-0002 8 Ch. Dig. Input 24V, 3ms, M12]
//         R3.Reamer[1].N30 (EP2028-0002) [EP2028-0002 8 Ch. Dig. Output 24V, 2A, M12]
//     R3.RT02 (EL6695-1001) [KRC4 secondary EL6695-1001]
//       modules: Module 1 (Sync Inputs), Module 2 (Safety Data (8 Byte)), Module 3 (Default IO)
//     ESW01.N01 (EP1908) [EP1908, 8 Ch. Safety Input 24V, TwinSAFE]
//       modules: Module 1 (FSOE)
//     R8.T01 (EK1100) [EK1100 EtherCAT Coupler (2A E-Bus)]
//       R8.T02 (EL6900) [EL6900, TwinSAFE PLC]
//       R8.T03 (EL1904) [EL1904, 4 Ch. Safety Input 24V, TwinSAFE]
//         modules: Module 1 (FSOES)
//       R8.T04 (EK1122) [EK1122 2 port EtherCAT junction]
//         R8.Reamer[1].N01 (EP1008-0002) [EP1008-0002 8 Ch. Dig. Input 24V, 3ms, M12]
//         R8.Reamer[1].N30 (EP2028-0002) [EP2028-0002 8 Ch. Dig. Output 24V, 2A, M12]
//     R8.RT02 (EL6695-1001) [KRC4 secondary EL6695-1001]
//       modules: Module 1 (Sync Inputs), Module 2 (Safety Data (8 Byte)), Module 3 (Default IO)
//     R9.T01 (EK1100) [EK1100 EtherCAT Coupler (2A E-Bus)]
//       R9.T02 (EL6900) [EL6900, TwinSAFE PLC]
//       R9.T03 (EL1904) [EL1904, 4 Ch. Safety Input 24V, TwinSAFE]
//         modules: Module 1 (FSOES)
//       R9.T04 (EK1122) [EK1122 2 port EtherCAT junction]
//         R9.Reamer[1].N01 (EP1008-0002) [EP1008-0002 8 Ch. Dig. Input 24V, 3ms, M12]
//         R9.Reamer[1].N30 (EP2028-0002) [EP2028-0002 8 Ch. Dig. Output 24V, 2A, M12]
//     R9.RT02 (EL6695-1001) [KRC4 secondary EL6695-1001]
//       modules: Module 1 (Sync Inputs), Module 2 (Safety Data (8 Byte)), Module 3 (Default IO)
//     R7.T01 (EK1100) [EK1100 EtherCAT Coupler (2A E-Bus)]
//       R7.T02 (EL6900) [EL6900, TwinSAFE PLC]
//       R7.T03 (EL1904) [EL1904, 4 Ch. Safety Input 24V, TwinSAFE]
//         modules: Module 1 (FSOES)
//       R7.T04 (EK1122) [EK1122 2 port EtherCAT junction]
//         R7.Reamer[1].N01 (EP1008-0002) [EP1008-0002 8 Ch. Dig. Input 24V, 3ms, M12]
//         R7.Reamer[1].N30 (EP2028-0002) [EP2028-0002 8 Ch. Dig. Output 24V, 2A, M12]
//     R7.RT02 (EL6695-1001) [KRC4 secondary EL6695-1001]
//       modules: Module 1 (Sync Inputs), Module 2 (Safety Data (8 Byte)), Module 3 (Default IO)
//     Fix01.N32_42 (EP1111-0000) [EP1111-0000 ID-Switch]
//     Fix01.N33_42 (EP1008-0002) [EP1008-0002 8 Ch. Dig. Input 24V, 3ms, M12]
//     Fix01.N34_43 (EP1111-0000) [EP1111-0000 ID-Switch]
//     Fix01.N35_43 (EP1008-0002) [EP1008-0002 8 Ch. Dig. Input 24V, 3ms, M12]
//     Fix01.N36_44 (EP1111-0000) [EP1111-0000 ID-Switch]
//     Fix01.N37_44 (EP1008-0002) [EP1008-0002 8 Ch. Dig. Input 24V, 3ms, M12]
//     Fix01.N38_45 (EP1111-0000) [EP1111-0000 ID-Switch]
//     Fix01.N39_45 (EP1008-0002) [EP1008-0002 8 Ch. Dig. Input 24V, 3ms, M12]
//     Fix01.N40_46 (EP1111-0000) [EP1111-0000 ID-Switch]
//     Fix01.N41_46 (EP1008-0002) [EP1008-0002 8 Ch. Dig. Input 24V, 3ms, M12]
//     Fix01.N42_47 (EP1111-0000) [EP1111-0000 ID-Switch]
//     Fix01.N43_47 (EP1008-0002) [EP1008-0002 8 Ch. Dig. Input 24V, 3ms, M12]
//     Fix02.N32_42 (EP1111-0000) [EP1111-0000 ID-Switch]
//     Fix02.N33_42 (EP1008-0002) [EP1008-0002 8 Ch. Dig. Input 24V, 3ms, M12]
//     Fix02.N34_43 (EP1111-0000) [EP1111-0000 ID-Switch]
//     Fix02.N35_43 (EP1008-0002) [EP1008-0002 8 Ch. Dig. Input 24V, 3ms, M12]
//     Fix02.N36_44 (EP1111-0000) [EP1111-0000 ID-Switch]
//     Fix02.N37_44 (EP1008-0002) [EP1008-0002 8 Ch. Dig. Input 24V, 3ms, M12]
//     Fix02.N38_45 (EP1111-0000) [EP1111-0000 ID-Switch]
//     Fix02.N39_45 (EP1008-0002) [EP1008-0002 8 Ch. Dig. Input 24V, 3ms, M12]
//     Fix02.N40_46 (EP1111-0000) [EP1111-0000 ID-Switch]
//     Fix02.N41_46 (EP1008-0002) [EP1008-0002 8 Ch. Dig. Input 24V, 3ms, M12]
//     Fix02.N42_47 (EP1111-0000) [EP1111-0000 ID-Switch]
//     Fix02.N43_47 (EP1008-0002) [EP1008-0002 8 Ch. Dig. Input 24V, 3ms, M12]
//   DEVICE PD01.T05 (EL6731) (disabled), AmsNetId 172.16.1.191.8.1
//     SIC01.N10 (GSD Box) (UNIGATE IC - Profibus) // Vendor: Deutschmann Automation GmbH Revision: V1.4
//     SIC01.N20 (GSD Box) (UNIGATE IC - Profibus) // Vendor: Deutschmann Automation GmbH Revision: V1.4
// variable links:
//   EtherCAT Master (EtherCAT) <-> EtherCAT Master (EtherCAT)/ESW01.N01 (EP1908)
//     IC01.T01 (EK1100)/IC01.T02 (EL6900)/ConnectionInputs/Message_9 TxPDO <-> Module 1 (FSOE)/FSOE Outputs/FSOE
//     IC01.T01 (EK1100)/IC01.T02 (EL6900)/ConnectionOutputs/Message_9 RxPDO <-> Module 1 (FSOE)/FSOE Inputs/FSOE
//   EtherCAT Master (EtherCAT) <-> EtherCAT Master (EtherCAT)/ESW02.N01 (EP1908)
//     IC01.T01 (EK1100)/IC01.T02 (EL6900)/ConnectionInputs/Message_10 TxPDO <-> Module 1 (FSOE)/FSOE Outputs/FSOE
//   EtherCAT Master (EtherCAT) <-> EtherCAT Master (EtherCAT)/ESW03.N01 (EP1908)
//     IC01.T01 (EK1100)/IC01.T02 (EL6900)/ConnectionOutputs/Message_11 RxPDO <-> Module 1 (FSOE)/FSOE Inputs/FSOE
//   EtherCAT Master (EtherCAT) <-> EtherCAT Master (EtherCAT)/IC01.T01 (EK1100)/IC01.T02 (EL6900)
//     ESW02.N01 (EP1908)/Module 1 (FSOE)/FSOE Inputs/FSOE <-> ConnectionOutputs/Message_10 RxPDO
//     ESW03.N01 (EP1908)/Module 1 (FSOE)/FSOE Outputs/FSOE <-> ConnectionInputs/Message_11 TxPDO
//     IC01.T01 (EK1100)/IC01.T03 (EL1904)/Module 1 (FSOES)/RxPDO/FSOE <-> ConnectionInputs/Message_1 TxPDO
//     IC01.T01 (EK1100)/IC01.T05 (EL1904)/Module 1 (FSOES)/RxPDO/FSOE <-> ConnectionInputs/Message_5 TxPDO
//     IC01.T01 (EK1100)/IC01.T07 (EL1904)/Module 1 (FSOES)/RxPDO/FSOE <-> ConnectionInputs/Message_6 TxPDO
//     IC01.T01 (EK1100)/IC01.T08 (EL1904)/Module 1 (FSOES)/RxPDO/FSOE <-> ConnectionInputs/Message_3 TxPDO
//     IC01.T01 (EK1100)/IC01.T09 (EL2904)/Module 1 (FSOES)/RxPDO/FSOE <-> ConnectionInputs/Message_7 TxPDO
//     IC01.T01 (EK1100)/IC01.T10 (EL2904)/Module 1 (FSOES)/RxPDO/FSOE <-> ConnectionInputs/Message_8 TxPDO
//     IC01.T01 (EK1100)/IC01.T03 (EL1904)/Module 1 (FSOES)/TxPDO/FSOE <-> ConnectionOutputs/Message_1 RxPDO
//     IC01.T01 (EK1100)/IC01.T04 (EL1904)/Module 1 (FSOES)/TxPDO/FSOE <-> ConnectionOutputs/Message_4 RxPDO
//     IC01.T01 (EK1100)/IC01.T06 (EL1904)/Module 1 (FSOES)/TxPDO/FSOE <-> ConnectionOutputs/Message_2 RxPDO
//     IC01.T01 (EK1100)/IC01.T07 (EL1904)/Module 1 (FSOES)/TxPDO/FSOE <-> ConnectionOutputs/Message_6 RxPDO
//     IC01.T01 (EK1100)/IC01.T10 (EL2904)/Module 1 (FSOES)/TxPDO/FSOE <-> ConnectionOutputs/Message_8 RxPDO
//     IC02.T01 (EK1100)/IC02.T02 (EL6900)/ConnectionInputs/Message_9 TxPDO <-> ConnectionOutputs/Message_12 RxPDO
//     IC02.T01 (EK1100)/IC02.T02 (EL6900)/ConnectionOutputs/Message_9 RxPDO <-> ConnectionInputs/Message_12 TxPDO
//     IS01.T01 (EK1100)/IS01.T02 (EL6900)/ConnectionInputs/Message_3 TxPDO <-> ConnectionOutputs/Message_43 RxPDO
//     MD01.N01 (EP1918-0002)/ConnectionOutputs/Message_8 RxPDO <-> ConnectionInputs/Message_105 TxPDO
//     MD02.N01 (EP1918-0002)/ConnectionOutputs/Message_8 RxPDO <-> ConnectionInputs/Message_106 TxPDO
//     MD02.N01 (EP1918-0002)/ConnectionInputs/Message_8 TxPDO <-> ConnectionOutputs/Message_106 RxPDO
//     R10.T01 (EK1100)/R10.T02 (EL6900)/ConnectionInputs/Message_2 TxPDO <-> ConnectionOutputs/Message_27 RxPDO
//     R2.T01 (EK1100)/R2.T02 (EL6900)/ConnectionInputs/Message_2 TxPDO <-> ConnectionOutputs/Message_19 RxPDO
//     R3.T01 (EK1100)/R3.T02 (EL6900)/ConnectionInputs/Message_2 TxPDO <-> ConnectionOutputs/Message_20 RxPDO
//     R4.T01 (EK1100)/R4.T02 (EL6900)/ConnectionInputs/Message_2 TxPDO <-> ConnectionOutputs/Message_21 RxPDO
//     R7.T01 (EK1100)/R7.T02 (EL6900)/ConnectionInputs/Message_2 TxPDO <-> ConnectionOutputs/Message_24 RxPDO
//     R9.T01 (EK1100)/R9.T02 (EL6900)/ConnectionInputs/Message_2 TxPDO <-> ConnectionOutputs/Message_26 RxPDO
//     R3.T01 (EK1100)/R3.T02 (EL6900)/ConnectionOutputs/Message_2 RxPDO <-> ConnectionInputs/Message_20 TxPDO
//     R5.T01 (EK1100)/R5.T02 (EL6900)/ConnectionOutputs/Message_2 RxPDO <-> ConnectionInputs/Message_22 TxPDO
//     R7.T01 (EK1100)/R7.T02 (EL6900)/ConnectionOutputs/Message_2 RxPDO <-> ConnectionInputs/Message_24 TxPDO
//     R8.T01 (EK1100)/R8.T02 (EL6900)/ConnectionOutputs/Message_2 RxPDO <-> ConnectionInputs/Message_25 TxPDO
//   EtherCAT Master (EtherCAT) <-> EtherCAT Master (EtherCAT)/IC01.T01 (EK1100)/IC01.T04 (EL1904)
//     IC01.T01 (EK1100)/IC01.T02 (EL6900)/ConnectionInputs/Message_4 TxPDO <-> Module 1 (FSOES)/RxPDO/FSOE
//   EtherCAT Master (EtherCAT) <-> EtherCAT Master (EtherCAT)/IC01.T01 (EK1100)/IC01.T05 (EL1904)
//     IC01.T01 (EK1100)/IC01.T02 (EL6900)/ConnectionOutputs/Message_5 RxPDO <-> Module 1 (FSOES)/TxPDO/FSOE
//   EtherCAT Master (EtherCAT) <-> EtherCAT Master (EtherCAT)/IC01.T01 (EK1100)/IC01.T06 (EL1904)
//     IC01.T01 (EK1100)/IC01.T02 (EL6900)/ConnectionInputs/Message_2 TxPDO <-> Module 1 (FSOES)/RxPDO/FSOE
//   EtherCAT Master (EtherCAT) <-> EtherCAT Master (EtherCAT)/IC01.T01 (EK1100)/IC01.T08 (EL1904)
//     IC01.T01 (EK1100)/IC01.T02 (EL6900)/ConnectionOutputs/Message_3 RxPDO <-> Module 1 (FSOES)/TxPDO/FSOE
//   EtherCAT Master (EtherCAT) <-> EtherCAT Master (EtherCAT)/IC01.T01 (EK1100)/IC01.T09 (EL2904)
//     IC01.T01 (EK1100)/IC01.T02 (EL6900)/ConnectionOutputs/Message_7 RxPDO <-> Module 1 (FSOES)/TxPDO/FSOE
//   EtherCAT Master (EtherCAT) <-> EtherCAT Master (EtherCAT)/IC02.T01 (EK1100)/IC02.T02 (EL6900)
//     IC02.T01 (EK1100)/IC02.T03 (EL1904)/Module 1 (FSOES)/TxPDO/FSOE <-> ConnectionOutputs/Message_1 RxPDO
//     IC02.T01 (EK1100)/IC02.T04 (EL1904)/Module 1 (FSOES)/TxPDO/FSOE <-> ConnectionOutputs/Message_3 RxPDO
//     IC02.T01 (EK1100)/IC02.T07 (EL1904)/Module 1 (FSOES)/TxPDO/FSOE <-> ConnectionOutputs/Message_4 RxPDO
//     IC02.T01 (EK1100)/IC02.T08 (EL1904)/Module 1 (FSOES)/TxPDO/FSOE <-> ConnectionOutputs/Message_6 RxPDO
//     IC02.T01 (EK1100)/IC02.T09 (EL2904)/Module 1 (FSOES)/TxPDO/FSOE <-> ConnectionOutputs/Message_7 RxPDO
//     IC02.T01 (EK1100)/IC02.T10 (EL2904)/Module 1 (FSOES)/TxPDO/FSOE <-> ConnectionOutputs/Message_8 RxPDO
//     IC02.T01 (EK1100)/IC02.T04 (EL1904)/Module 1 (FSOES)/RxPDO/FSOE <-> ConnectionInputs/Message_3 TxPDO
//     IC02.T01 (EK1100)/IC02.T08 (EL1904)/Module 1 (FSOES)/RxPDO/FSOE <-> ConnectionInputs/Message_6 TxPDO
//     IC02.T01 (EK1100)/IC02.T09 (EL2904)/Module 1 (FSOES)/RxPDO/FSOE <-> ConnectionInputs/Message_7 TxPDO
//   EtherCAT Master (EtherCAT) <-> EtherCAT Master (EtherCAT)/IC02.T01 (EK1100)/IC02.T03 (EL1904)
//     IC02.T01 (EK1100)/IC02.T02 (EL6900)/ConnectionInputs/Message_1 TxPDO <-> Module 1 (FSOES)/RxPDO/FSOE
//   EtherCAT Master (EtherCAT) <-> EtherCAT Master (EtherCAT)/IC02.T01 (EK1100)/IC02.T05 (EL1904)
//     IC02.T01 (EK1100)/IC02.T02 (EL6900)/ConnectionInputs/Message_5 TxPDO <-> Module 1 (FSOES)/RxPDO/FSOE
//     IC02.T01 (EK1100)/IC02.T02 (EL6900)/ConnectionOutputs/Message_5 RxPDO <-> Module 1 (FSOES)/TxPDO/FSOE
//   EtherCAT Master (EtherCAT) <-> EtherCAT Master (EtherCAT)/IC02.T01 (EK1100)/IC02.T06 (EL1904)
//     IC02.T01 (EK1100)/IC02.T02 (EL6900)/ConnectionInputs/Message_2 TxPDO <-> Module 1 (FSOES)/RxPDO/FSOE
//     IC02.T01 (EK1100)/IC02.T02 (EL6900)/ConnectionOutputs/Message_2 RxPDO <-> Module 1 (FSOES)/TxPDO/FSOE
//   EtherCAT Master (EtherCAT) <-> EtherCAT Master (EtherCAT)/IC02.T01 (EK1100)/IC02.T07 (EL1904)
//     IC02.T01 (EK1100)/IC02.T02 (EL6900)/ConnectionInputs/Message_4 TxPDO <-> Module 1 (FSOES)/RxPDO/FSOE
//   EtherCAT Master (EtherCAT) <-> EtherCAT Master (EtherCAT)/IC02.T01 (EK1100)/IC02.T10 (EL2904)
//     IC02.T01 (EK1100)/IC02.T02 (EL6900)/ConnectionInputs/Message_8 TxPDO <-> Module 1 (FSOES)/RxPDO/FSOE
//   EtherCAT Master (EtherCAT) <-> EtherCAT Master (EtherCAT)/IC03.T01 (EK1100)/IC03.T02 (EL6900)
//     IC01.T01 (EK1100)/IC01.T02 (EL6900)/ConnectionInputs/Message_13 TxPDO <-> ConnectionOutputs/Message_9 RxPDO
//     IC01.T01 (EK1100)/IC01.T02 (EL6900)/ConnectionOutputs/Message_13 RxPDO <-> ConnectionInputs/Message_9 TxPDO
//     IC03.T01 (EK1100)/IC03.T03 (EL1904)/Module 1 (FSOES)/RxPDO/FSOE <-> ConnectionInputs/Message_1 TxPDO
//     IC03.T01 (EK1100)/IC03.T04 (EL1904)/Module 1 (FSOES)/RxPDO/FSOE <-> ConnectionInputs/Message_4 TxPDO
//     IC03.T01 (EK1100)/IC03.T08 (EL1904)/Module 1 (FSOES)/RxPDO/FSOE <-> ConnectionInputs/Message_3 TxPDO
//     IC03.T01 (EK1100)/IC03.T09 (EL2904)/Module 1 (FSOES)/RxPDO/FSOE <-> ConnectionInputs/Message_7 TxPDO
//     IC03.T01 (EK1100)/IC03.T03 (EL1904)/Module 1 (FSOES)/TxPDO/FSOE <-> ConnectionOutputs/Message_1 RxPDO
//     IC03.T01 (EK1100)/IC03.T04 (EL1904)/Module 1 (FSOES)/TxPDO/FSOE <-> ConnectionOutputs/Message_4 RxPDO
//     IC03.T01 (EK1100)/IC03.T08 (EL1904)/Module 1 (FSOES)/TxPDO/FSOE <-> ConnectionOutputs/Message_3 RxPDO
//     IC03.T01 (EK1100)/IC03.T10 (EL2904)/Module 1 (FSOES)/TxPDO/FSOE <-> ConnectionOutputs/Message_8 RxPDO
//   EtherCAT Master (EtherCAT) <-> EtherCAT Master (EtherCAT)/IC03.T01 (EK1100)/IC03.T05 (EL1904)
//     IC03.T01 (EK1100)/IC03.T02 (EL6900)/ConnectionInputs/Message_5 TxPDO <-> Module 1 (FSOES)/RxPDO/FSOE
//     IC03.T01 (EK1100)/IC03.T02 (EL6900)/ConnectionOutputs/Message_5 RxPDO <-> Module 1 (FSOES)/TxPDO/FSOE
//   EtherCAT Master (EtherCAT) <-> EtherCAT Master (EtherCAT)/IC03.T01 (EK1100)/IC03.T06 (EL1904)
//     IC03.T01 (EK1100)/IC03.T02 (EL6900)/ConnectionInputs/Message_2 TxPDO <-> Module 1 (FSOES)/RxPDO/FSOE
//     IC03.T01 (EK1100)/IC03.T02 (EL6900)/ConnectionOutputs/Message_2 RxPDO <-> Module 1 (FSOES)/TxPDO/FSOE
//   EtherCAT Master (EtherCAT) <-> EtherCAT Master (EtherCAT)/IC03.T01 (EK1100)/IC03.T09 (EL2904)
//     IC03.T01 (EK1100)/IC03.T02 (EL6900)/ConnectionOutputs/Message_7 RxPDO <-> Module 1 (FSOES)/TxPDO/FSOE
//   EtherCAT Master (EtherCAT) <-> EtherCAT Master (EtherCAT)/IC03.T01 (EK1100)/IC03.T10 (EL2904)
//     IC03.T01 (EK1100)/IC03.T02 (EL6900)/ConnectionInputs/Message_8 TxPDO <-> Module 1 (FSOES)/RxPDO/FSOE
//   EtherCAT Master (EtherCAT) <-> EtherCAT Master (EtherCAT)/IS01.T01 (EK1100)/IS01.T02 (EL6900)
//     IC01.T01 (EK1100)/IC01.T02 (EL6900)/ConnectionInputs/Message_43 TxPDO <-> ConnectionOutputs/Message_3 RxPDO
//     IS01.T01 (EK1100)/IS01.T03 (EL1904)/Module 1 (FSOES)/TxPDO/FSOE <-> ConnectionOutputs/Message_2 RxPDO
//     IS01.T01 (EK1100)/IS01.T04 (EL2904)/Module 1 (FSOES)/TxPDO/FSOE <-> ConnectionOutputs/Message_1 RxPDO
//   EtherCAT Master (EtherCAT) <-> EtherCAT Master (EtherCAT)/IS01.T01 (EK1100)/IS01.T03 (EL1904)
//     IS01.T01 (EK1100)/IS01.T02 (EL6900)/ConnectionInputs/Message_2 TxPDO <-> Module 1 (FSOES)/RxPDO/FSOE
//   EtherCAT Master (EtherCAT) <-> EtherCAT Master (EtherCAT)/IS01.T01 (EK1100)/IS01.T04 (EL2904)
//     IS01.T01 (EK1100)/IS01.T02 (EL6900)/ConnectionInputs/Message_1 TxPDO <-> Module 1 (FSOES)/RxPDO/FSOE
//   EtherCAT Master (EtherCAT) <-> EtherCAT Master (EtherCAT)/MD01.N01 (EP1918-0002)
//     IC01.T01 (EK1100)/IC01.T02 (EL6900)/ConnectionOutputs/Message_105 RxPDO <-> ConnectionInputs/Message_8 TxPDO
//   EtherCAT Master (EtherCAT) <-> EtherCAT Master (EtherCAT)/R1.RT02 (EL6695-1001)
//     R1.T01 (EK1100)/R1.T02 (EL6900)/ConnectionOutputs/Message_1 RxPDO <-> Module 2 (Safety Data (8 Byte))/Inputs/FSOE
//   EtherCAT Master (EtherCAT) <-> EtherCAT Master (EtherCAT)/R1.T01 (EK1100)/R1.T02 (EL6900)
//     IC01.T01 (EK1100)/IC01.T02 (EL6900)/ConnectionInputs/Message_18 TxPDO <-> ConnectionOutputs/Message_2 RxPDO
//     IC01.T01 (EK1100)/IC01.T02 (EL6900)/ConnectionOutputs/Message_18 RxPDO <-> ConnectionInputs/Message_2 TxPDO
//     R1.RT02 (EL6695-1001)/Module 2 (Safety Data (8 Byte))/Outputs/FSOE <-> ConnectionInputs/Message_1 TxPDO
//     R1.T01 (EK1100)/R1.T03 (EL1904)/Module 1 (FSOES)/RxPDO/FSOE <-> ConnectionInputs/Message_24 TxPDO
//   EtherCAT Master (EtherCAT) <-> EtherCAT Master (EtherCAT)/R1.T01 (EK1100)/R1.T03 (EL1904)
//     R1.T01 (EK1100)/R1.T02 (EL6900)/ConnectionOutputs/Message_24 RxPDO <-> Module 1 (FSOES)/TxPDO/FSOE
//   EtherCAT Master (EtherCAT) <-> EtherCAT Master (EtherCAT)/R10.T01 (EK1100)/R10.T02 (EL6900)
//     IC01.T01 (EK1100)/IC01.T02 (EL6900)/ConnectionInputs/Message_27 TxPDO <-> ConnectionOutputs/Message_2 RxPDO
//     R10.RT02 (EL6695-1001)/Module 2 (Safety Data (8 Byte))/Inputs/FSOE <-> ConnectionOutputs/Message_1 RxPDO
//     R10.RT02 (EL6695-1001)/Module 2 (Safety Data (8 Byte))/Outputs/FSOE <-> ConnectionInputs/Message_1 TxPDO
//   EtherCAT Master (EtherCAT) <-> EtherCAT Master (EtherCAT)/R11.RT02 (EL6695-1001)
//     R11.T01 (EK1100)/R11.T02 (EL6900)/ConnectionInputs/Message_1 TxPDO <-> Module 2 (Safety Data (8 Byte))/Outputs/FSOE
//   EtherCAT Master (EtherCAT) <-> EtherCAT Master (EtherCAT)/R11.T01 (EK1100)/R11.T02 (EL6900)
//     IC01.T01 (EK1100)/IC01.T02 (EL6900)/ConnectionInputs/Message_28 TxPDO <-> ConnectionOutputs/Message_2 RxPDO
//     IC01.T01 (EK1100)/IC01.T02 (EL6900)/ConnectionOutputs/Message_28 RxPDO <-> ConnectionInputs/Message_2 TxPDO
//     R11.RT02 (EL6695-1001)/Module 2 (Safety Data (8 Byte))/Inputs/FSOE <-> ConnectionOutputs/Message_1 RxPDO
//   EtherCAT Master (EtherCAT) <-> EtherCAT Master (EtherCAT)/R2.RT02 (EL6695-1001)
//     R2.T01 (EK1100)/R2.T02 (EL6900)/ConnectionOutputs/Message_1 RxPDO <-> Module 2 (Safety Data (8 Byte))/Inputs/FSOE
//   EtherCAT Master (EtherCAT) <-> EtherCAT Master (EtherCAT)/R2.T01 (EK1100)/R2.T02 (EL6900)
//     IC01.T01 (EK1100)/IC01.T02 (EL6900)/ConnectionInputs/Message_19 TxPDO <-> ConnectionOutputs/Message_2 RxPDO
//     R2.RT02 (EL6695-1001)/Module 2 (Safety Data (8 Byte))/Outputs/FSOE <-> ConnectionInputs/Message_1 TxPDO
//   EtherCAT Master (EtherCAT) <-> EtherCAT Master (EtherCAT)/R3.RT02 (EL6695-1001)
//     R3.T01 (EK1100)/R3.T02 (EL6900)/ConnectionInputs/Message_1 TxPDO <-> Module 2 (Safety Data (8 Byte))/Outputs/FSOE
//   EtherCAT Master (EtherCAT) <-> EtherCAT Master (EtherCAT)/R3.T01 (EK1100)/R3.T02 (EL6900)
//     R3.RT02 (EL6695-1001)/Module 2 (Safety Data (8 Byte))/Inputs/FSOE <-> ConnectionOutputs/Message_1 RxPDO
//   EtherCAT Master (EtherCAT) <-> EtherCAT Master (EtherCAT)/R4.RT02 (EL6695-1001)
//     R4.T01 (EK1100)/R4.T02 (EL6900)/ConnectionInputs/Message_1 TxPDO <-> Module 2 (Safety Data (8 Byte))/Outputs/FSOE
//     R4.T01 (EK1100)/R4.T02 (EL6900)/ConnectionOutputs/Message_1 RxPDO <-> Module 2 (Safety Data (8 Byte))/Inputs/FSOE
//   EtherCAT Master (EtherCAT) <-> EtherCAT Master (EtherCAT)/R4.T01 (EK1100)/R4.T02 (EL6900)
//     IC01.T01 (EK1100)/IC01.T02 (EL6900)/ConnectionInputs/Message_21 TxPDO <-> ConnectionOutputs/Message_2 RxPDO
//   EtherCAT Master (EtherCAT) <-> EtherCAT Master (EtherCAT)/R5.T01 (EK1100)/R5.T02 (EL6900)
//     IC01.T01 (EK1100)/IC01.T02 (EL6900)/ConnectionOutputs/Message_22 RxPDO <-> ConnectionInputs/Message_2 TxPDO
//     R5.RT02 (EL6695-1001)/Module 2 (Safety Data (8 Byte))/Inputs/FSOE <-> ConnectionOutputs/Message_1 RxPDO
//     R5.RT02 (EL6695-1001)/Module 2 (Safety Data (8 Byte))/Outputs/FSOE <-> ConnectionInputs/Message_1 TxPDO
//     R5.T01 (EK1100)/R5.T03 (EL1904)/Module 1 (FSOES)/RxPDO/FSOE <-> ConnectionInputs/Message_22 TxPDO
//   EtherCAT Master (EtherCAT) <-> EtherCAT Master (EtherCAT)/R5.T01 (EK1100)/R5.T03 (EL1904)
//     R5.T01 (EK1100)/R5.T02 (EL6900)/ConnectionOutputs/Message_22 RxPDO <-> Module 1 (FSOES)/TxPDO/FSOE
//   EtherCAT Master (EtherCAT) <-> EtherCAT Master (EtherCAT)/R6.T01 (EK1100)/R6.T02 (EL6900)
//     IC01.T01 (EK1100)/IC01.T02 (EL6900)/ConnectionInputs/Message_23 TxPDO <-> ConnectionOutputs/Message_2 RxPDO
//     IC01.T01 (EK1100)/IC01.T02 (EL6900)/ConnectionOutputs/Message_23 RxPDO <-> ConnectionInputs/Message_2 TxPDO
//     R6.RT02 (EL6695-1001)/Module 2 (Safety Data (8 Byte))/Inputs/FSOE <-> ConnectionOutputs/Message_1 RxPDO
//     R6.RT02 (EL6695-1001)/Module 2 (Safety Data (8 Byte))/Outputs/FSOE <-> ConnectionInputs/Message_1 TxPDO
//   EtherCAT Master (EtherCAT) <-> EtherCAT Master (EtherCAT)/R7.RT02 (EL6695-1001)
//     R7.T01 (EK1100)/R7.T02 (EL6900)/ConnectionInputs/Message_1 TxPDO <-> Module 2 (Safety Data (8 Byte))/Outputs/FSOE
//   EtherCAT Master (EtherCAT) <-> EtherCAT Master (EtherCAT)/R7.T01 (EK1100)/R7.T02 (EL6900)
//     R7.RT02 (EL6695-1001)/Module 2 (Safety Data (8 Byte))/Inputs/FSOE <-> ConnectionOutputs/Message_1 RxPDO
//   EtherCAT Master (EtherCAT) <-> EtherCAT Master (EtherCAT)/R8.T01 (EK1100)/R8.T02 (EL6900)
//     IC01.T01 (EK1100)/IC01.T02 (EL6900)/ConnectionOutputs/Message_25 RxPDO <-> ConnectionInputs/Message_2 TxPDO
//     R8.RT02 (EL6695-1001)/Module 2 (Safety Data (8 Byte))/Inputs/FSOE <-> ConnectionOutputs/Message_1 RxPDO
//     R8.RT02 (EL6695-1001)/Module 2 (Safety Data (8 Byte))/Outputs/FSOE <-> ConnectionInputs/Message_1 TxPDO
//   EtherCAT Master (EtherCAT) <-> EtherCAT Master (EtherCAT)/R9.RT02 (EL6695-1001)
//     R9.T01 (EK1100)/R9.T02 (EL6900)/ConnectionInputs/Message_1 TxPDO <-> Module 2 (Safety Data (8 Byte))/Outputs/FSOE
//   EtherCAT Master (EtherCAT) <-> EtherCAT Master (EtherCAT)/R9.T01 (EK1100)/R9.T02 (EL6900)
//     IC01.T01 (EK1100)/IC01.T02 (EL6900)/ConnectionInputs/Message_26 TxPDO <-> ConnectionOutputs/Message_2 RxPDO
//     R9.RT02 (EL6695-1001)/Module 2 (Safety Data (8 Byte))/Inputs/FSOE <-> ConnectionOutputs/Message_1 RxPDO
//   EtherCAT Master (EtherCAT) <-> EtherCAT Master (EtherCAT)/SS01.N01 (EP9128-0021)/VertiGuard.N02 (EP1908)
//     IC02.T01 (EK1100)/IC02.T02 (EL6900)/ConnectionInputs/Message_31 TxPDO <-> Module 1 (FSOE)/FSOE Outputs/FSOE
//     IC02.T01 (EK1100)/IC02.T02 (EL6900)/ConnectionOutputs/Message_31 RxPDO <-> Module 1 (FSOE)/FSOE Inputs/FSOE
//   SODG11_SSCC610_2403701_PLC/SODG11_SSCC610_2403701_PLC Instance <-> EtherCAT Master (EtherCAT)
//     Standard Inputs/MAIN.ECAT_Master.HW_Status/DevState <-> Inputs/DevState
//     Standard Inputs/MAIN.ECAT_Master.HW_Status/Frm0State <-> Inputs/Frm0State
//     Standard Inputs/MAIN.ECAT_Master.HW_Status/Frm0WcState <-> Inputs/Frm0WcState
//     Standard Inputs/MAIN.ECAT_Master.HW_Status/Infodata/AmsNetId <-> InfoData/AmsNetId
//     Standard Inputs/MAIN.ECAT_Master.HW_Status/Infodata/CfgSlaveCount <-> InfoData/CfgSlaveCount
//     Standard Inputs/MAIN.ECAT_Master.HW_Status/Infodata/ChangeCount <-> InfoData/ChangeCount
//     Standard Inputs/MAIN.ECAT_Master.HW_Status/Infodata/DevID <-> InfoData/DevId
//     Standard Inputs/MAIN.ECAT_Master.HW_Status/SlaveCount <-> Inputs/SlaveCount
//   SODG11_SSCC610_2403701_PLC/SODG11_SSCC610_2403701_PLC Instance <-> EtherCAT Master (EtherCAT)/ESW01.N01 (EP1908)
//     Standard Inputs/MAIN.ESW01.N01/I <-> Module 1 (FSOE)/FSOE Inputs/FSOE/InputChannel1
//     Standard Inputs/MAIN.ESW01.N01/I @bit 1 <-> Module 1 (FSOE)/FSOE Inputs/FSOE/InputChannel2
//     Standard Inputs/MAIN.ESW01.N01/I @bit 2 <-> Module 1 (FSOE)/FSOE Inputs/FSOE/InputChannel3
//     Standard Inputs/MAIN.ESW01.N01/I @bit 3 <-> Module 1 (FSOE)/FSOE Inputs/FSOE/InputChannel4
//     Standard Inputs/MAIN.ESW01.N01/I @bit 4 <-> Module 1 (FSOE)/FSOE Inputs/FSOE/InputChannel5
//     Standard Inputs/MAIN.ESW01.N01/I @bit 5 <-> Module 1 (FSOE)/FSOE Inputs/FSOE/InputChannel6
//     Standard Inputs/MAIN.ESW01.N01/I @bit 6 <-> Module 1 (FSOE)/FSOE Inputs/FSOE/InputChannel7
//     Standard Inputs/MAIN.ESW01.N01/I @bit 7 <-> Module 1 (FSOE)/FSOE Inputs/FSOE/InputChannel8
//     Standard Inputs/MAIN.ESW01.N01/InfoData/State <-> InfoData/State
//   SODG11_SSCC610_2403701_PLC/SODG11_SSCC610_2403701_PLC Instance <-> EtherCAT Master (EtherCAT)/ESW02.N01 (EP1908)
//     Standard Inputs/MAIN.ESW02.N01/I <-> Module 1 (FSOE)/FSOE Inputs/FSOE/InputChannel1
//     Standard Inputs/MAIN.ESW02.N01/I @bit 1 <-> Module 1 (FSOE)/FSOE Inputs/FSOE/InputChannel2
//     Standard Inputs/MAIN.ESW02.N01/I @bit 2 <-> Module 1 (FSOE)/FSOE Inputs/FSOE/InputChannel3
//     Standard Inputs/MAIN.ESW02.N01/I @bit 3 <-> Module 1 (FSOE)/FSOE Inputs/FSOE/InputChannel4
//     Standard Inputs/MAIN.ESW02.N01/I @bit 4 <-> Module 1 (FSOE)/FSOE Inputs/FSOE/InputChannel5
//     Standard Inputs/MAIN.ESW02.N01/I @bit 5 <-> Module 1 (FSOE)/FSOE Inputs/FSOE/InputChannel6
//     Standard Inputs/MAIN.ESW02.N01/I @bit 6 <-> Module 1 (FSOE)/FSOE Inputs/FSOE/InputChannel7
//     Standard Inputs/MAIN.ESW02.N01/I @bit 7 <-> Module 1 (FSOE)/FSOE Inputs/FSOE/InputChannel8
//     Standard Inputs/MAIN.ESW02.N01/InfoData/State <-> InfoData/State
//   SODG11_SSCC610_2403701_PLC/SODG11_SSCC610_2403701_PLC Instance <-> EtherCAT Master (EtherCAT)/ESW03.N01 (EP1908)
//     Standard Inputs/MAIN.ESW03.N01/I <-> Module 1 (FSOE)/FSOE Inputs/FSOE/InputChannel1
//     Standard Inputs/MAIN.ESW03.N01/I @bit 1 <-> Module 1 (FSOE)/FSOE Inputs/FSOE/InputChannel2
//     Standard Inputs/MAIN.ESW03.N01/I @bit 2 <-> Module 1 (FSOE)/FSOE Inputs/FSOE/InputChannel3
//     Standard Inputs/MAIN.ESW03.N01/I @bit 3 <-> Module 1 (FSOE)/FSOE Inputs/FSOE/InputChannel4
//     Standard Inputs/MAIN.ESW03.N01/I @bit 4 <-> Module 1 (FSOE)/FSOE Inputs/FSOE/InputChannel5
//     Standard Inputs/MAIN.ESW03.N01/I @bit 5 <-> Module 1 (FSOE)/FSOE Inputs/FSOE/InputChannel6
//     Standard Inputs/MAIN.ESW03.N01/I @bit 6 <-> Module 1 (FSOE)/FSOE Inputs/FSOE/InputChannel7
//     Standard Inputs/MAIN.ESW03.N01/I @bit 7 <-> Module 1 (FSOE)/FSOE Inputs/FSOE/InputChannel8
//     Standard Inputs/MAIN.ESW03.N01/InfoData/State <-> InfoData/State
//   SODG11_SSCC610_2403701_PLC/SODG11_SSCC610_2403701_PLC Instance <-> EtherCAT Master (EtherCAT)/Fix01.N32_42 (EP1111-0000)
//     Standard Inputs/Fix01.N32/ID <-> ID Inputs/ID
//     Standard Inputs/Fix01.N32/InfoData/State <-> InfoData/State
//     Standard Inputs/Fix01.N32/Wc_State <-> WcState/WcState
//   SODG11_SSCC610_2403701_PLC/SODG11_SSCC610_2403701_PLC Instance <-> EtherCAT Master (EtherCAT)/Fix01.N33_42 (EP1008-0002)
//     Standard Inputs/Fix01.N33/I <-> Channel 1/Input
//     Standard Inputs/Fix01.N33/I @bit 1 <-> Channel 2/Input
//     Standard Inputs/Fix01.N33/I @bit 2 <-> Channel 3/Input
//     Standard Inputs/Fix01.N33/I @bit 3 <-> Channel 4/Input
//     Standard Inputs/Fix01.N33/I @bit 4 <-> Channel 5/Input
//     Standard Inputs/Fix01.N33/I @bit 5 <-> Channel 6/Input
//     Standard Inputs/Fix01.N33/I @bit 6 <-> Channel 7/Input
//     Standard Inputs/Fix01.N33/I @bit 7 <-> Channel 8/Input
//     Standard Inputs/Fix01.N33/InfoData/State <-> InfoData/State
//     Standard Inputs/Fix01.N33/Wc_State <-> WcState/WcState
//   SODG11_SSCC610_2403701_PLC/SODG11_SSCC610_2403701_PLC Instance <-> EtherCAT Master (EtherCAT)/Fix01.N34_43 (EP1111-0000)
//     Standard Inputs/Fix01.N34/ID <-> ID Inputs/ID
//     Standard Inputs/Fix01.N34/InfoData/State <-> InfoData/State
//     Standard Inputs/Fix01.N34/Wc_State <-> WcState/WcState
//   SODG11_SSCC610_2403701_PLC/SODG11_SSCC610_2403701_PLC Instance <-> EtherCAT Master (EtherCAT)/Fix01.N35_43 (EP1008-0002)
//     Standard Inputs/Fix01.N35/I <-> Channel 1/Input
//     Standard Inputs/Fix01.N35/I @bit 1 <-> Channel 2/Input
//     Standard Inputs/Fix01.N35/I @bit 2 <-> Channel 3/Input
//     Standard Inputs/Fix01.N35/I @bit 3 <-> Channel 4/Input
//     Standard Inputs/Fix01.N35/I @bit 4 <-> Channel 5/Input
//     Standard Inputs/Fix01.N35/I @bit 5 <-> Channel 6/Input
//     Standard Inputs/Fix01.N35/I @bit 6 <-> Channel 7/Input
//     Standard Inputs/Fix01.N35/I @bit 7 <-> Channel 8/Input
//     Standard Inputs/Fix01.N35/InfoData/State <-> InfoData/State
//     Standard Inputs/Fix01.N35/Wc_State <-> WcState/WcState
//   SODG11_SSCC610_2403701_PLC/SODG11_SSCC610_2403701_PLC Instance <-> EtherCAT Master (EtherCAT)/Fix01.N36_44 (EP1111-0000)
//     Standard Inputs/Fix01.N36/ID <-> ID Inputs/ID
//     Standard Inputs/Fix01.N36/InfoData/State <-> InfoData/State
//     Standard Inputs/Fix01.N36/Wc_State <-> WcState/WcState
//   SODG11_SSCC610_2403701_PLC/SODG11_SSCC610_2403701_PLC Instance <-> EtherCAT Master (EtherCAT)/Fix01.N37_44 (EP1008-0002)
//     Standard Inputs/Fix01.N37/I <-> Channel 1/Input
//     Standard Inputs/Fix01.N37/I @bit 1 <-> Channel 2/Input
//     Standard Inputs/Fix01.N37/I @bit 2 <-> Channel 3/Input
//     Standard Inputs/Fix01.N37/I @bit 3 <-> Channel 4/Input
//     Standard Inputs/Fix01.N37/I @bit 4 <-> Channel 5/Input
//     Standard Inputs/Fix01.N37/I @bit 5 <-> Channel 6/Input
//     Standard Inputs/Fix01.N37/I @bit 6 <-> Channel 7/Input
//     Standard Inputs/Fix01.N37/I @bit 7 <-> Channel 8/Input
//     Standard Inputs/Fix01.N37/InfoData/State <-> InfoData/State
//     Standard Inputs/Fix01.N37/Wc_State <-> WcState/WcState
//   SODG11_SSCC610_2403701_PLC/SODG11_SSCC610_2403701_PLC Instance <-> EtherCAT Master (EtherCAT)/Fix01.N38_45 (EP1111-0000)
//     Standard Inputs/Fix01.N38/ID <-> ID Inputs/ID
//     Standard Inputs/Fix01.N38/InfoData/State <-> InfoData/State
//     Standard Inputs/Fix01.N38/Wc_State <-> WcState/WcState
//   SODG11_SSCC610_2403701_PLC/SODG11_SSCC610_2403701_PLC Instance <-> EtherCAT Master (EtherCAT)/Fix01.N39_45 (EP1008-0002)
//     Standard Inputs/Fix01.N39/I <-> Channel 1/Input
//     Standard Inputs/Fix01.N39/I @bit 1 <-> Channel 2/Input
//     Standard Inputs/Fix01.N39/I @bit 2 <-> Channel 3/Input
//     Standard Inputs/Fix01.N39/I @bit 3 <-> Channel 4/Input
//     Standard Inputs/Fix01.N39/I @bit 4 <-> Channel 5/Input
//     Standard Inputs/Fix01.N39/I @bit 5 <-> Channel 6/Input
//     Standard Inputs/Fix01.N39/I @bit 6 <-> Channel 7/Input
//     Standard Inputs/Fix01.N39/I @bit 7 <-> Channel 8/Input
//     Standard Inputs/Fix01.N39/InfoData/State <-> InfoData/State
//     Standard Inputs/Fix01.N39/Wc_State <-> WcState/WcState
//   SODG11_SSCC610_2403701_PLC/SODG11_SSCC610_2403701_PLC Instance <-> EtherCAT Master (EtherCAT)/Fix01.N40_46 (EP1111-0000)
//     Standard Inputs/Fix01.N40/ID <-> ID Inputs/ID
//     Standard Inputs/Fix01.N40/InfoData/State <-> InfoData/State
//     Standard Inputs/Fix01.N40/Wc_State <-> WcState/WcState
//   SODG11_SSCC610_2403701_PLC/SODG11_SSCC610_2403701_PLC Instance <-> EtherCAT Master (EtherCAT)/Fix01.N41_46 (EP1008-0002)
//     Standard Inputs/Fix01.N41/I <-> Channel 1/Input
//     Standard Inputs/Fix01.N41/I @bit 1 <-> Channel 2/Input
//     Standard Inputs/Fix01.N41/I @bit 2 <-> Channel 3/Input
//     Standard Inputs/Fix01.N41/I @bit 3 <-> Channel 4/Input
//     Standard Inputs/Fix01.N41/I @bit 4 <-> Channel 5/Input
//     Standard Inputs/Fix01.N41/I @bit 5 <-> Channel 6/Input
//     Standard Inputs/Fix01.N41/I @bit 6 <-> Channel 7/Input
//     Standard Inputs/Fix01.N41/I @bit 7 <-> Channel 8/Input
//     Standard Inputs/Fix01.N41/InfoData/State <-> InfoData/State
//     Standard Inputs/Fix01.N41/Wc_State <-> WcState/WcState
//   SODG11_SSCC610_2403701_PLC/SODG11_SSCC610_2403701_PLC Instance <-> EtherCAT Master (EtherCAT)/Fix01.N42_47 (EP1111-0000)
//     Standard Inputs/Fix01.N42/ID <-> ID Inputs/ID
//     Standard Inputs/Fix01.N42/InfoData/State <-> InfoData/State
//     Standard Inputs/Fix01.N42/Wc_State <-> WcState/WcState
//   SODG11_SSCC610_2403701_PLC/SODG11_SSCC610_2403701_PLC Instance <-> EtherCAT Master (EtherCAT)/Fix01.N43_47 (EP1008-0002)
//     Standard Inputs/Fix01.N43/I <-> Channel 1/Input
//     Standard Inputs/Fix01.N43/I @bit 1 <-> Channel 2/Input
//     Standard Inputs/Fix01.N43/I @bit 2 <-> Channel 3/Input
//     Standard Inputs/Fix01.N43/I @bit 3 <-> Channel 4/Input
//     Standard Inputs/Fix01.N43/I @bit 4 <-> Channel 5/Input
//     Standard Inputs/Fix01.N43/I @bit 5 <-> Channel 6/Input
//     Standard Inputs/Fix01.N43/I @bit 6 <-> Channel 7/Input
//     Standard Inputs/Fix01.N43/I @bit 7 <-> Channel 8/Input
//     Standard Inputs/Fix01.N43/InfoData/State <-> InfoData/State
//     Standard Inputs/Fix01.N43/Wc_State <-> WcState/WcState
//   SODG11_SSCC610_2403701_PLC/SODG11_SSCC610_2403701_PLC Instance <-> EtherCAT Master (EtherCAT)/Fix02.N32_42 (EP1111-0000)
//     Standard Inputs/Fix02.N32/ID <-> ID Inputs/ID
//     Standard Inputs/Fix02.N32/InfoData/State <-> InfoData/State
//     Standard Inputs/Fix02.N32/Wc_State <-> WcState/WcState
//   SODG11_SSCC610_2403701_PLC/SODG11_SSCC610_2403701_PLC Instance <-> EtherCAT Master (EtherCAT)/Fix02.N33_42 (EP1008-0002)
//     Standard Inputs/Fix02.N33/I <-> Channel 1/Input
//     Standard Inputs/Fix02.N33/I @bit 1 <-> Channel 2/Input
//     Standard Inputs/Fix02.N33/I @bit 2 <-> Channel 3/Input
//     Standard Inputs/Fix02.N33/I @bit 3 <-> Channel 4/Input
//     Standard Inputs/Fix02.N33/I @bit 4 <-> Channel 5/Input
//     Standard Inputs/Fix02.N33/I @bit 5 <-> Channel 6/Input
//     Standard Inputs/Fix02.N33/I @bit 6 <-> Channel 7/Input
//     Standard Inputs/Fix02.N33/I @bit 7 <-> Channel 8/Input
//     Standard Inputs/Fix02.N33/InfoData/State <-> InfoData/State
//     Standard Inputs/Fix02.N33/Wc_State <-> WcState/WcState
//   SODG11_SSCC610_2403701_PLC/SODG11_SSCC610_2403701_PLC Instance <-> EtherCAT Master (EtherCAT)/Fix02.N34_43 (EP1111-0000)
//     Standard Inputs/Fix02.N34/ID <-> ID Inputs/ID
//     Standard Inputs/Fix02.N34/InfoData/State <-> InfoData/State
//     Standard Inputs/Fix02.N34/Wc_State <-> WcState/WcState
//   SODG11_SSCC610_2403701_PLC/SODG11_SSCC610_2403701_PLC Instance <-> EtherCAT Master (EtherCAT)/Fix02.N35_43 (EP1008-0002)
//     Standard Inputs/Fix02.N35/I <-> Channel 1/Input
//     Standard Inputs/Fix02.N35/I @bit 1 <-> Channel 2/Input
//     Standard Inputs/Fix02.N35/I @bit 2 <-> Channel 3/Input
//     Standard Inputs/Fix02.N35/I @bit 3 <-> Channel 4/Input
//     Standard Inputs/Fix02.N35/I @bit 4 <-> Channel 5/Input
//     Standard Inputs/Fix02.N35/I @bit 5 <-> Channel 6/Input
//     Standard Inputs/Fix02.N35/I @bit 6 <-> Channel 7/Input
//     Standard Inputs/Fix02.N35/I @bit 7 <-> Channel 8/Input
//     Standard Inputs/Fix02.N35/InfoData/State <-> InfoData/State
//     Standard Inputs/Fix02.N35/Wc_State <-> WcState/WcState
//   SODG11_SSCC610_2403701_PLC/SODG11_SSCC610_2403701_PLC Instance <-> EtherCAT Master (EtherCAT)/Fix02.N36_44 (EP1111-0000)
//     Standard Inputs/Fix02.N36/ID <-> ID Inputs/ID
//     Standard Inputs/Fix02.N36/InfoData/State <-> InfoData/State
//     Standard Inputs/Fix02.N36/Wc_State <-> WcState/WcState
//   SODG11_SSCC610_2403701_PLC/SODG11_SSCC610_2403701_PLC Instance <-> EtherCAT Master (EtherCAT)/Fix02.N37_44 (EP1008-0002)
//     Standard Inputs/Fix02.N37/I <-> Channel 1/Input
//     Standard Inputs/Fix02.N37/I @bit 1 <-> Channel 2/Input
//     Standard Inputs/Fix02.N37/I @bit 2 <-> Channel 3/Input
//     Standard Inputs/Fix02.N37/I @bit 3 <-> Channel 4/Input
//     Standard Inputs/Fix02.N37/I @bit 4 <-> Channel 5/Input
//     Standard Inputs/Fix02.N37/I @bit 5 <-> Channel 6/Input
//     Standard Inputs/Fix02.N37/I @bit 6 <-> Channel 7/Input
//     Standard Inputs/Fix02.N37/I @bit 7 <-> Channel 8/Input
//     Standard Inputs/Fix02.N37/InfoData/State <-> InfoData/State
//     Standard Inputs/Fix02.N37/Wc_State <-> WcState/WcState
//   SODG11_SSCC610_2403701_PLC/SODG11_SSCC610_2403701_PLC Instance <-> EtherCAT Master (EtherCAT)/Fix02.N38_45 (EP1111-0000)
//     Standard Inputs/Fix02.N38/ID <-> ID Inputs/ID
//     Standard Inputs/Fix02.N38/InfoData/State <-> InfoData/State
//     Standard Inputs/Fix02.N38/Wc_State <-> WcState/WcState
//   SODG11_SSCC610_2403701_PLC/SODG11_SSCC610_2403701_PLC Instance <-> EtherCAT Master (EtherCAT)/Fix02.N39_45 (EP1008-0002)
//     Standard Inputs/Fix02.N39/I <-> Channel 1/Input
//     Standard Inputs/Fix02.N39/I @bit 1 <-> Channel 2/Input
//     Standard Inputs/Fix02.N39/I @bit 2 <-> Channel 3/Input
//     Standard Inputs/Fix02.N39/I @bit 3 <-> Channel 4/Input
//     Standard Inputs/Fix02.N39/I @bit 4 <-> Channel 5/Input
//     Standard Inputs/Fix02.N39/I @bit 5 <-> Channel 6/Input
//     Standard Inputs/Fix02.N39/I @bit 6 <-> Channel 7/Input
//     Standard Inputs/Fix02.N39/I @bit 7 <-> Channel 8/Input
//     Standard Inputs/Fix02.N39/InfoData/State <-> InfoData/State
//     Standard Inputs/Fix02.N39/Wc_State <-> WcState/WcState
//   SODG11_SSCC610_2403701_PLC/SODG11_SSCC610_2403701_PLC Instance <-> EtherCAT Master (EtherCAT)/Fix02.N40_46 (EP1111-0000)
//     Standard Inputs/Fix02.N40/ID <-> ID Inputs/ID
//     Standard Inputs/Fix02.N40/InfoData/State <-> InfoData/State
//     Standard Inputs/Fix02.N40/Wc_State <-> WcState/WcState
//   SODG11_SSCC610_2403701_PLC/SODG11_SSCC610_2403701_PLC Instance <-> EtherCAT Master (EtherCAT)/Fix02.N41_46 (EP1008-0002)
//     Standard Inputs/Fix02.N41/I <-> Channel 1/Input
//     Standard Inputs/Fix02.N41/I @bit 1 <-> Channel 2/Input
//     Standard Inputs/Fix02.N41/I @bit 2 <-> Channel 3/Input
//     Standard Inputs/Fix02.N41/I @bit 3 <-> Channel 4/Input
//     Standard Inputs/Fix02.N41/I @bit 4 <-> Channel 5/Input
//     Standard Inputs/Fix02.N41/I @bit 5 <-> Channel 6/Input
//     Standard Inputs/Fix02.N41/I @bit 6 <-> Channel 7/Input
//     Standard Inputs/Fix02.N41/I @bit 7 <-> Channel 8/Input
//     Standard Inputs/Fix02.N41/InfoData/State <-> InfoData/State
//     Standard Inputs/Fix02.N41/Wc_State <-> WcState/WcState
//   SODG11_SSCC610_2403701_PLC/SODG11_SSCC610_2403701_PLC Instance <-> EtherCAT Master (EtherCAT)/Fix02.N42_47 (EP1111-0000)
//     Standard Inputs/Fix02.N42/ID <-> ID Inputs/ID
//     Standard Inputs/Fix02.N42/InfoData/State <-> InfoData/State
//     Standard Inputs/Fix02.N42/Wc_State <-> WcState/WcState
//   SODG11_SSCC610_2403701_PLC/SODG11_SSCC610_2403701_PLC Instance <-> EtherCAT Master (EtherCAT)/Fix02.N43_47 (EP1008-0002)
//     Standard Inputs/Fix02.N43/I <-> Channel 1/Input
//     Standard Inputs/Fix02.N43/I @bit 1 <-> Channel 2/Input
//     Standard Inputs/Fix02.N43/I @bit 2 <-> Channel 3/Input
//     Standard Inputs/Fix02.N43/I @bit 3 <-> Channel 4/Input
//     Standard Inputs/Fix02.N43/I @bit 4 <-> Channel 5/Input
//     Standard Inputs/Fix02.N43/I @bit 5 <-> Channel 6/Input
//     Standard Inputs/Fix02.N43/I @bit 6 <-> Channel 7/Input
//     Standard Inputs/Fix02.N43/I @bit 7 <-> Channel 8/Input
//     Standard Inputs/Fix02.N43/InfoData/State <-> InfoData/State
//     Standard Inputs/Fix02.N43/Wc_State <-> WcState/WcState
//   SODG11_SSCC610_2403701_PLC/SODG11_SSCC610_2403701_PLC Instance <-> EtherCAT Master (EtherCAT)/IC01.T01 (EK1100)
//     Standard Inputs/MAIN.IC01.T01/InfoData/State <-> InfoData/State
//   SODG11_SSCC610_2403701_PLC/SODG11_SSCC610_2403701_PLC Instance <-> EtherCAT Master (EtherCAT)/IC01.T01 (EK1100)/IC01.T02 (EL6900)
//     Standard Inputs/MAIN.Access_Violation_IC01 <-> StandardInputs/Standard Out Var 108
//     Standard Inputs/MAIN.All_Estops_OK <-> StandardInputs/Standard Out Var 78
//     Standard Inputs/MAIN.All_SafetyGates_OK <-> StandardInputs/Standard Out Var 77
//     Standard Inputs/MAIN.IC01.T02_STAT/Device_Info_Data/Project_CRC <-> Device Info Data/Project CRC
//     Standard Inputs/MAIN.IC01.T02_STAT/FBs_FB_ERR <-> StandardInputs/Standard Out Var 79
//     Standard Inputs/MAIN.IC01.T02_STAT/FBs_FB_ERR @bit 1 <-> StandardInputs/Standard Out Var 80
//     Standard Inputs/MAIN.IC01.T02_STAT/FBs_FB_ERR @bit 2 <-> StandardInputs/Standard Out Var 81
//     Standard Inputs/MAIN.IC01.T02_STAT/FBs_FB_ERR @bit 8 <-> StandardInputs/Standard Out Var 82
//     Standard Inputs/MAIN.IC01.T02_STAT/FBs_FB_ERR @bit 16 <-> StandardInputs/Standard Out Var 83
//     Standard Inputs/MAIN.IC01.T02_STAT/FBs_FB_ERR @bit 17 <-> StandardInputs/Standard Out Var 84
//     Standard Inputs/MAIN.IC01.T02_STAT/FBs_FB_ERR @bit 24 <-> StandardInputs/Standard Out Var 85
//     Standard Inputs/MAIN.IC01.T02_STAT/FBs_FB_ERR @bit 25 <-> StandardInputs/Standard Out Var 86
//     Standard Inputs/MAIN.IC01.T02_STAT/FBs_FB_ERR @bit 26 <-> StandardInputs/Standard Out Var 87
//     Standard Inputs/MAIN.IC01.T02_STAT/InfoData/AdsAddr/netId <-> InfoData/AdsAddr/netId
//     Standard Inputs/MAIN.IC01.T02_STAT/InfoData/AdsAddr/port <-> InfoData/AdsAddr/port
//     Standard Inputs/MAIN.IC01.T02_STAT/InfoData/State <-> InfoData/State
//     Standard Inputs/MAIN.IC01.T02_STAT/SGs_COM_ERR @bit 5 <-> StandardInputs/Standard Out Var 100
//     Standard Inputs/MAIN.IC01.T02_STAT/SGs_COM_ERR @bit 1 <-> StandardInputs/Standard Out Var 62
//     Standard Inputs/MAIN.IC01.T02_STAT/SGs_COM_ERR @bit 2 <-> StandardInputs/Standard Out Var 69
//     Standard Inputs/MAIN.IC01.T02_STAT/SGs_COM_ERR @bit 4 <-> StandardInputs/Standard Out Var 75
//     Standard Inputs/MAIN.IC01.T02_STAT/SGs_COM_ERR <-> StandardInputs/Standard Out Var 59
//     Standard Inputs/MAIN.IC01.T02_STAT/SGs_FB_ERR @bit 5 <-> StandardInputs/Standard Out Var 101
//     Standard Inputs/MAIN.IC01.T02_STAT/SGs_FB_ERR @bit 1 <-> StandardInputs/Standard Out Var 61
//     Standard Inputs/MAIN.IC01.T02_STAT/SGs_FB_ERR @bit 2 <-> StandardInputs/Standard Out Var 64
//     Standard Inputs/MAIN.IC01.T02_STAT/SGs_FB_ERR @bit 4 <-> StandardInputs/Standard Out Var 74
//     Standard Inputs/MAIN.IC01.T02_STAT/SGs_FB_ERR <-> StandardInputs/Standard Out Var 58
//     Standard Inputs/MAIN.IC01.T02_STAT/SGs_OUT_ERR @bit 5 <-> StandardInputs/Standard Out Var 102
//     Standard Inputs/MAIN.IC01.T02_STAT/SGs_OUT_ERR @bit 1 <-> StandardInputs/Standard Out Var 63
//     Standard Inputs/MAIN.IC01.T02_STAT/SGs_OUT_ERR @bit 2 <-> StandardInputs/Standard Out Var 70
//     Standard Inputs/MAIN.IC01.T02_STAT/SGs_OUT_ERR @bit 4 <-> StandardInputs/Standard Out Var 76
//     Standard Inputs/MAIN.IC01.T02_STAT/SGs_OUT_ERR <-> StandardInputs/Standard Out Var 60
//     Standard Inputs/MAIN.IC01.T09/Q <-> StandardInputs/Standard Out Var 65
//     Standard Inputs/MAIN.IC01.T10/Q <-> StandardInputs/Standard Out Var 67
//     Standard Inputs/MAIN.IC01.T09/Q @bit 1 <-> StandardInputs/Standard Out Var 66
//     Standard Inputs/MAIN.IC01.T10/Q @bit 1 <-> StandardInputs/Standard Out Var 68
//     Standard Outputs/MAIN.IC01.T02_CMD/FBs_ControlPowerPB <-> StandardOutputs/Standard In Var 50
//     Standard Outputs/MAIN.IC01.T02_CMD/SGs_ERRAck <-> StandardOutputs/Standard In Var 45
//     Standard Outputs/MAIN.IC01.T02_CMD/SGs_ERRAck <-> StandardOutputs/Standard In Var 47
//     Standard Outputs/MAIN.IC01.T02_CMD/SGs_ERRAck <-> StandardOutputs/Standard In Var 49
//     Standard Outputs/MAIN.IC01.T02_CMD/SGs_ERRAck <-> StandardOutputs/Standard In Var 57
//     Standard Outputs/MAIN.IC01.T02_CMD/SGs_ERRAck <-> StandardOutputs/Standard In Var 98
//     Standard Outputs/MAIN.IC01.T02_CMD/SGs_RUNSTOP <-> StandardOutputs/Standard In Var 44
//     Standard Outputs/MAIN.IC01.T02_CMD/SGs_RUNSTOP <-> StandardOutputs/Standard In Var 46
//     Standard Outputs/MAIN.IC01.T02_CMD/SGs_RUNSTOP <-> StandardOutputs/Standard In Var 48
//     Standard Outputs/MAIN.IC01.T02_CMD/SGs_RUNSTOP <-> StandardOutputs/Standard In Var 56
//     Standard Outputs/MAIN.IC01.T02_CMD/SGs_RUNSTOP <-> StandardOutputs/Standard In Var 99
//   SODG11_SSCC610_2403701_PLC/SODG11_SSCC610_2403701_PLC Instance <-> EtherCAT Master (EtherCAT)/IC01.T01 (EK1100)/IC01.T03 (EL1904)
//     Standard Inputs/MAIN.IC01.T03/I <-> Module 1 (FSOES)/TxPDO/FSOE/InputChannel1
//     Standard Inputs/MAIN.IC01.T03/I @bit 1 <-> Module 1 (FSOES)/TxPDO/FSOE/InputChannel2
//     Standard Inputs/MAIN.IC01.T03/I @bit 2 <-> Module 1 (FSOES)/TxPDO/FSOE/InputChannel3
//     Standard Inputs/MAIN.IC01.T03/I @bit 3 <-> Module 1 (FSOES)/TxPDO/FSOE/InputChannel4
//     Standard Inputs/MAIN.IC01.T03/InfoData/State <-> InfoData/State
//   SODG11_SSCC610_2403701_PLC/SODG11_SSCC610_2403701_PLC Instance <-> EtherCAT Master (EtherCAT)/IC01.T01 (EK1100)/IC01.T04 (EL1904)
//     Standard Inputs/MAIN.IC01.T04/I <-> Module 1 (FSOES)/TxPDO/FSOE/InputChannel1
//     Standard Inputs/MAIN.IC01.T04/I @bit 1 <-> Module 1 (FSOES)/TxPDO/FSOE/InputChannel2
//     Standard Inputs/MAIN.IC01.T04/I @bit 2 <-> Module 1 (FSOES)/TxPDO/FSOE/InputChannel3
//     Standard Inputs/MAIN.IC01.T04/I @bit 3 <-> Module 1 (FSOES)/TxPDO/FSOE/InputChannel4
//     Standard Inputs/MAIN.IC01.T04/InfoData/State <-> InfoData/State
//   SODG11_SSCC610_2403701_PLC/SODG11_SSCC610_2403701_PLC Instance <-> EtherCAT Master (EtherCAT)/IC01.T01 (EK1100)/IC01.T05 (EL1904)
//     Standard Inputs/MAIN.IC01.T05/I <-> Module 1 (FSOES)/TxPDO/FSOE/InputChannel1
//     Standard Inputs/MAIN.IC01.T05/I @bit 1 <-> Module 1 (FSOES)/TxPDO/FSOE/InputChannel2
//     Standard Inputs/MAIN.IC01.T05/I @bit 2 <-> Module 1 (FSOES)/TxPDO/FSOE/InputChannel3
//     Standard Inputs/MAIN.IC01.T05/I @bit 3 <-> Module 1 (FSOES)/TxPDO/FSOE/InputChannel4
//     Standard Inputs/MAIN.IC01.T05/InfoData/State <-> InfoData/State
//   SODG11_SSCC610_2403701_PLC/SODG11_SSCC610_2403701_PLC Instance <-> EtherCAT Master (EtherCAT)/IC01.T01 (EK1100)/IC01.T06 (EL1904)
//     Standard Inputs/MAIN.IC01.T06/I <-> Module 1 (FSOES)/TxPDO/FSOE/InputChannel1
//     Standard Inputs/MAIN.IC01.T06/I @bit 1 <-> Module 1 (FSOES)/TxPDO/FSOE/InputChannel2
//     Standard Inputs/MAIN.IC01.T06/I @bit 2 <-> Module 1 (FSOES)/TxPDO/FSOE/InputChannel3
//     Standard Inputs/MAIN.IC01.T06/I @bit 3 <-> Module 1 (FSOES)/TxPDO/FSOE/InputChannel4
//     Standard Inputs/MAIN.IC01.T06/InfoData/State <-> InfoData/State
//   SODG11_SSCC610_2403701_PLC/SODG11_SSCC610_2403701_PLC Instance <-> EtherCAT Master (EtherCAT)/IC01.T01 (EK1100)/IC01.T07 (EL1904)
//     Standard Inputs/MAIN.IC01.T07/I <-> Module 1 (FSOES)/TxPDO/FSOE/InputChannel1
//     Standard Inputs/MAIN.IC01.T07/I @bit 1 <-> Module 1 (FSOES)/TxPDO/FSOE/InputChannel2
//     Standard Inputs/MAIN.IC01.T07/I @bit 2 <-> Module 1 (FSOES)/TxPDO/FSOE/InputChannel3
//     Standard Inputs/MAIN.IC01.T07/I @bit 3 <-> Module 1 (FSOES)/TxPDO/FSOE/InputChannel4
//     Standard Inputs/MAIN.IC01.T07/InfoData/State <-> InfoData/State
//   SODG11_SSCC610_2403701_PLC/SODG11_SSCC610_2403701_PLC Instance <-> EtherCAT Master (EtherCAT)/IC01.T01 (EK1100)/IC01.T08 (EL1904)
//     Standard Inputs/MAIN.IC01.T08/I <-> Module 1 (FSOES)/TxPDO/FSOE/InputChannel1
//     Standard Inputs/MAIN.IC01.T08/I @bit 1 <-> Module 1 (FSOES)/TxPDO/FSOE/InputChannel2
//     Standard Inputs/MAIN.IC01.T08/I @bit 2 <-> Module 1 (FSOES)/TxPDO/FSOE/InputChannel3
//     Standard Inputs/MAIN.IC01.T08/I @bit 3 <-> Module 1 (FSOES)/TxPDO/FSOE/InputChannel4
//     Standard Inputs/MAIN.IC01.T08/InfoData/State <-> InfoData/State
//   SODG11_SSCC610_2403701_PLC/SODG11_SSCC610_2403701_PLC Instance <-> EtherCAT Master (EtherCAT)/IC01.T01 (EK1100)/IC01.T09 (EL2904)
//     Standard Inputs/MAIN.IC01.T09/InfoData/State <-> InfoData/State
//   SODG11_SSCC610_2403701_PLC/SODG11_SSCC610_2403701_PLC Instance <-> EtherCAT Master (EtherCAT)/IC01.T01 (EK1100)/IC01.T10 (EL2904)
//     Standard Inputs/MAIN.IC01.T10/InfoData/State <-> InfoData/State
//   SODG11_SSCC610_2403701_PLC/SODG11_SSCC610_2403701_PLC Instance <-> EtherCAT Master (EtherCAT)/IC01.T01 (EK1100)/IC01.T11 (EL9410)
//     Standard Inputs/MAIN.IC01.T11/InfoData/State <-> InfoData/State
//     Standard Inputs/MAIN.IC01.T11/Up_UnderVoltage <-> Status Up/Undervoltage
//     Standard Inputs/MAIN.IC01.T11/Us_Undervoltage <-> Status Us/Undervoltage
//     Standard Inputs/MAIN.IC01.T11/WcState <-> WcState/WcState
//   SODG11_SSCC610_2403701_PLC/SODG11_SSCC610_2403701_PLC Instance <-> EtherCAT Master (EtherCAT)/IC01.T01 (EK1100)/IC01.T12 (EL1004)
//     Standard Inputs/MAIN.IC01.T12/I <-> Channel 1/Input
//     Standard Inputs/MAIN.IC01.T12/I @bit 1 <-> Channel 2/Input
//     Standard Inputs/MAIN.IC01.T12/I @bit 2 <-> Channel 3/Input
//     Standard Inputs/MAIN.IC01.T12/I @bit 3 <-> Channel 4/Input
//     Standard Inputs/MAIN.IC01.T12/InfoData/State <-> InfoData/State
//   SODG11_SSCC610_2403701_PLC/SODG11_SSCC610_2403701_PLC Instance <-> EtherCAT Master (EtherCAT)/IC01.T01 (EK1100)/IC01.T13 (EL1004)
//     Standard Inputs/MAIN.IC01.T13/I <-> Channel 1/Input
//     Standard Inputs/MAIN.IC01.T13/I @bit 1 <-> Channel 2/Input
//     Standard Inputs/MAIN.IC01.T13/I @bit 2 <-> Channel 3/Input
//     Standard Inputs/MAIN.IC01.T13/I @bit 3 <-> Channel 4/Input
//     Standard Inputs/MAIN.IC01.T13/InfoData/State <-> InfoData/State
//   SODG11_SSCC610_2403701_PLC/SODG11_SSCC610_2403701_PLC Instance <-> EtherCAT Master (EtherCAT)/IC01.T01 (EK1100)/IC01.T14 (EL2008)
//     Standard Inputs/MAIN.IC01.T14_STAT/InfoData/State <-> InfoData/State
//     Standard Outputs/MAIN.IC01.T14/Q <-> Channel 1/Output
//     Standard Outputs/MAIN.IC01.T14/Q @bit 1 <-> Channel 2/Output
//     Standard Outputs/MAIN.IC01.T14/Q @bit 2 <-> Channel 3/Output
//     Standard Outputs/MAIN.IC01.T14/Q @bit 3 <-> Channel 4/Output
//     Standard Outputs/MAIN.IC01.T14/Q @bit 4 <-> Channel 5/Output
//     Standard Outputs/MAIN.IC01.T14/Q @bit 5 <-> Channel 6/Output
//     Standard Outputs/MAIN.IC01.T14/Q @bit 6 <-> Channel 7/Output
//     Standard Outputs/MAIN.IC01.T14/Q @bit 7 <-> Channel 8/Output
//   SODG11_SSCC610_2403701_PLC/SODG11_SSCC610_2403701_PLC Instance <-> EtherCAT Master (EtherCAT)/IC01.T01 (EK1100)/IC01.T15 (EL2622)
//     Standard Inputs/MAIN.IC01.T15_STAT/InfoData/State <-> InfoData/State
//     Standard Outputs/MAIN.IC01.T15/Q0 <-> Channel 1/Output
//     Standard Outputs/MAIN.IC01.T15/Q1 <-> Channel 2/Output
//   SODG11_SSCC610_2403701_PLC/SODG11_SSCC610_2403701_PLC Instance <-> EtherCAT Master (EtherCAT)/IC01.T01 (EK1100)/IC01.T16 (EK1122)
//     Standard Inputs/MAIN.IC01.T16/InfoData/State <-> InfoData/State
//   SODG11_SSCC610_2403701_PLC/SODG11_SSCC610_2403701_PLC Instance <-> EtherCAT Master (EtherCAT)/IC01.T01 (EK1100)/IC01.T16 (EK1122)/Fix01.N01 (EP1008-0002)
//     Standard Inputs/Fix01.N01/I <-> Channel 1/Input
//     Standard Inputs/Fix01.N01/I @bit 1 <-> Channel 2/Input
//     Standard Inputs/Fix01.N01/I @bit 2 <-> Channel 3/Input
//     Standard Inputs/Fix01.N01/I @bit 3 <-> Channel 4/Input
//     Standard Inputs/Fix01.N01/I @bit 4 <-> Channel 5/Input
//     Standard Inputs/Fix01.N01/I @bit 5 <-> Channel 6/Input
//     Standard Inputs/Fix01.N01/I @bit 6 <-> Channel 7/Input
//     Standard Inputs/Fix01.N01/I @bit 7 <-> Channel 8/Input
//     Standard Inputs/Fix01.N01/InfoData/State <-> InfoData/State
//     Standard Inputs/Fix01.N01/Wc_State <-> WcState/WcState
//   SODG11_SSCC610_2403701_PLC/SODG11_SSCC610_2403701_PLC Instance <-> EtherCAT Master (EtherCAT)/IC01.T01 (EK1100)/IC01.T16 (EK1122)/Fix01.N02 (EP1008-0002)
//     Standard Inputs/Fix01.N02/I <-> Channel 1/Input
//     Standard Inputs/Fix01.N02/I @bit 1 <-> Channel 2/Input
//     Standard Inputs/Fix01.N02/I @bit 2 <-> Channel 3/Input
//     Standard Inputs/Fix01.N02/I @bit 3 <-> Channel 4/Input
//     Standard Inputs/Fix01.N02/I @bit 4 <-> Channel 5/Input
//     Standard Inputs/Fix01.N02/I @bit 5 <-> Channel 6/Input
//     Standard Inputs/Fix01.N02/I @bit 6 <-> Channel 7/Input
//     Standard Inputs/Fix01.N02/I @bit 7 <-> Channel 8/Input
//     Standard Inputs/Fix01.N02/InfoData/State <-> InfoData/State
//     Standard Inputs/Fix01.N02/Wc_State <-> WcState/WcState
//   SODG11_SSCC610_2403701_PLC/SODG11_SSCC610_2403701_PLC Instance <-> EtherCAT Master (EtherCAT)/IC01.T01 (EK1100)/IC01.T16 (EK1122)/Fix01.N03 (EP1008-0002)
//     Standard Inputs/Fix01.N03/I <-> Channel 1/Input
//     Standard Inputs/Fix01.N03/I @bit 1 <-> Channel 2/Input
//     Standard Inputs/Fix01.N03/I @bit 2 <-> Channel 3/Input
//     Standard Inputs/Fix01.N03/I @bit 3 <-> Channel 4/Input
//     Standard Inputs/Fix01.N03/I @bit 4 <-> Channel 5/Input
//     Standard Inputs/Fix01.N03/I @bit 5 <-> Channel 6/Input
//     Standard Inputs/Fix01.N03/I @bit 6 <-> Channel 7/Input
//     Standard Inputs/Fix01.N03/I @bit 7 <-> Channel 8/Input
//     Standard Inputs/Fix01.N03/InfoData/State <-> InfoData/State
//     Standard Inputs/Fix01.N03/Wc_State <-> WcState/WcState
//   SODG11_SSCC610_2403701_PLC/SODG11_SSCC610_2403701_PLC Instance <-> EtherCAT Master (EtherCAT)/IC01.T01 (EK1100)/IC01.T16 (EK1122)/Fix01.N04 (EP1008-0002)
//     Standard Inputs/Fix01.N04/I <-> Channel 1/Input
//     Standard Inputs/Fix01.N04/I @bit 1 <-> Channel 2/Input
//     Standard Inputs/Fix01.N04/I @bit 2 <-> Channel 3/Input
//     Standard Inputs/Fix01.N04/I @bit 3 <-> Channel 4/Input
//     Standard Inputs/Fix01.N04/I @bit 4 <-> Channel 5/Input
//     Standard Inputs/Fix01.N04/I @bit 5 <-> Channel 6/Input
//     Standard Inputs/Fix01.N04/I @bit 6 <-> Channel 7/Input
//     Standard Inputs/Fix01.N04/I @bit 7 <-> Channel 8/Input
//     Standard Inputs/Fix01.N04/InfoData/State <-> InfoData/State
//     Standard Inputs/Fix01.N04/Wc_State <-> WcState/WcState
//   SODG11_SSCC610_2403701_PLC/SODG11_SSCC610_2403701_PLC Instance <-> EtherCAT Master (EtherCAT)/IC01.T01 (EK1100)/IC01.T16 (EK1122)/Fix01.N05 (EP1008-0002)
//     Standard Inputs/Fix01.N05/I <-> Channel 1/Input
//     Standard Inputs/Fix01.N05/I @bit 1 <-> Channel 2/Input
//     Standard Inputs/Fix01.N05/I @bit 2 <-> Channel 3/Input
//     Standard Inputs/Fix01.N05/I @bit 3 <-> Channel 4/Input
//     Standard Inputs/Fix01.N05/I @bit 4 <-> Channel 5/Input
//     Standard Inputs/Fix01.N05/I @bit 5 <-> Channel 6/Input
//     Standard Inputs/Fix01.N05/I @bit 6 <-> Channel 7/Input
//     Standard Inputs/Fix01.N05/I @bit 7 <-> Channel 8/Input
//     Standard Inputs/Fix01.N05/InfoData/State <-> InfoData/State
//     Standard Inputs/Fix01.N05/Wc_State <-> WcState/WcState
//   SODG11_SSCC610_2403701_PLC/SODG11_SSCC610_2403701_PLC Instance <-> EtherCAT Master (EtherCAT)/IC01.T01 (EK1100)/IC01.T16 (EK1122)/Fix01.N06 (EP1008-0002)
//     Standard Inputs/Fix01.N06/I <-> Channel 1/Input
//     Standard Inputs/Fix01.N06/I @bit 1 <-> Channel 2/Input
//     Standard Inputs/Fix01.N06/I @bit 2 <-> Channel 3/Input
//     Standard Inputs/Fix01.N06/I @bit 3 <-> Channel 4/Input
//     Standard Inputs/Fix01.N06/I @bit 4 <-> Channel 5/Input
//     Standard Inputs/Fix01.N06/I @bit 5 <-> Channel 6/Input
//     Standard Inputs/Fix01.N06/I @bit 6 <-> Channel 7/Input
//     Standard Inputs/Fix01.N06/I @bit 7 <-> Channel 8/Input
//     Standard Inputs/Fix01.N06/InfoData/State <-> InfoData/State
//     Standard Inputs/Fix01.N06/Wc_State <-> WcState/WcState
//   SODG11_SSCC610_2403701_PLC/SODG11_SSCC610_2403701_PLC Instance <-> EtherCAT Master (EtherCAT)/IC01.T01 (EK1100)/IC01.T16 (EK1122)/Fix01.N07 (EP1008-0002)
//     Standard Inputs/Fix01.N07/I <-> Channel 1/Input
//     Standard Inputs/Fix01.N07/I @bit 1 <-> Channel 2/Input
//     Standard Inputs/Fix01.N07/I @bit 2 <-> Channel 3/Input
//     Standard Inputs/Fix01.N07/I @bit 3 <-> Channel 4/Input
//     Standard Inputs/Fix01.N07/I @bit 4 <-> Channel 5/Input
//     Standard Inputs/Fix01.N07/I @bit 5 <-> Channel 6/Input
//     Standard Inputs/Fix01.N07/I @bit 6 <-> Channel 7/Input
//     Standard Inputs/Fix01.N07/I @bit 7 <-> Channel 8/Input
//     Standard Inputs/Fix01.N07/InfoData/State <-> InfoData/State
//     Standard Inputs/Fix01.N07/Wc_State <-> WcState/WcState
//   SODG11_SSCC610_2403701_PLC/SODG11_SSCC610_2403701_PLC Instance <-> EtherCAT Master (EtherCAT)/IC01.T01 (EK1100)/IC01.T16 (EK1122)/Fix01.N08 (EP1008-0002)
//     Standard Inputs/Fix01.N08/I <-> Channel 1/Input
//     Standard Inputs/Fix01.N08/I @bit 1 <-> Channel 2/Input
//     Standard Inputs/Fix01.N08/I @bit 2 <-> Channel 3/Input
//     Standard Inputs/Fix01.N08/I @bit 3 <-> Channel 4/Input
//     Standard Inputs/Fix01.N08/I @bit 4 <-> Channel 5/Input
//     Standard Inputs/Fix01.N08/I @bit 5 <-> Channel 6/Input
//     Standard Inputs/Fix01.N08/I @bit 6 <-> Channel 7/Input
//     Standard Inputs/Fix01.N08/I @bit 7 <-> Channel 8/Input
//     Standard Inputs/Fix01.N08/InfoData/State <-> InfoData/State
//     Standard Inputs/Fix01.N08/Wc_State <-> WcState/WcState
//   SODG11_SSCC610_2403701_PLC/SODG11_SSCC610_2403701_PLC Instance <-> EtherCAT Master (EtherCAT)/IC01.T01 (EK1100)/IC01.T16 (EK1122)/Fix01.N09 (EP1008-0002)
//     Standard Inputs/Fix01.N09/I <-> Channel 1/Input
//     Standard Inputs/Fix01.N09/I @bit 1 <-> Channel 2/Input
//     Standard Inputs/Fix01.N09/I @bit 2 <-> Channel 3/Input
//     Standard Inputs/Fix01.N09/I @bit 3 <-> Channel 4/Input
//     Standard Inputs/Fix01.N09/I @bit 4 <-> Channel 5/Input
//     Standard Inputs/Fix01.N09/I @bit 5 <-> Channel 6/Input
//     Standard Inputs/Fix01.N09/I @bit 6 <-> Channel 7/Input
//     Standard Inputs/Fix01.N09/I @bit 7 <-> Channel 8/Input
//     Standard Inputs/Fix01.N09/InfoData/State <-> InfoData/State
//     Standard Inputs/Fix01.N09/Wc_State <-> WcState/WcState
//   SODG11_SSCC610_2403701_PLC/SODG11_SSCC610_2403701_PLC Instance <-> EtherCAT Master (EtherCAT)/IC01.T01 (EK1100)/IC01.T16 (EK1122)/Fix01.N10 (EP1008-0002)
//     Standard Inputs/Fix01.N10/I <-> Channel 1/Input
//     Standard Inputs/Fix01.N10/I @bit 1 <-> Channel 2/Input
//     Standard Inputs/Fix01.N10/I @bit 2 <-> Channel 3/Input
//     Standard Inputs/Fix01.N10/I @bit 3 <-> Channel 4/Input
//     Standard Inputs/Fix01.N10/I @bit 4 <-> Channel 5/Input
//     Standard Inputs/Fix01.N10/I @bit 5 <-> Channel 6/Input
//     Standard Inputs/Fix01.N10/I @bit 6 <-> Channel 7/Input
//     Standard Inputs/Fix01.N10/I @bit 7 <-> Channel 8/Input
//     Standard Inputs/Fix01.N10/InfoData/State <-> InfoData/State
//     Standard Inputs/Fix01.N10/Wc_State <-> WcState/WcState
//   SODG11_SSCC610_2403701_PLC/SODG11_SSCC610_2403701_PLC Instance <-> EtherCAT Master (EtherCAT)/IC01.T01 (EK1100)/IC01.T16 (EK1122)/Fix01.N100 (EX260-SEC1)
//     Standard Inputs/Fix01.N100_STAT/InfoData/State <-> InfoData/State
//     Standard Outputs/Fix01.N100/Q <-> Byte 0/Output
//     Standard Outputs/Fix01.N100/Q @bit 8 <-> Byte 1/Output
//     Standard Outputs/Fix01.N100/Q @bit 16 <-> Byte 2/Output
//     Standard Outputs/Fix01.N100/Q @bit 24 <-> Byte 3/Output
//   SODG11_SSCC610_2403701_PLC/SODG11_SSCC610_2403701_PLC Instance <-> EtherCAT Master (EtherCAT)/IC01.T01 (EK1100)/IC01.T16 (EK1122)/Fix01.N101 (EX260-SEC1)
//     Standard Inputs/Fix01.N101_STAT/InfoData/State <-> InfoData/State
//     Standard Outputs/Fix01.N101/Q <-> Byte 0/Output
//     Standard Outputs/Fix01.N101/Q @bit 8 <-> Byte 1/Output
//     Standard Outputs/Fix01.N101/Q @bit 16 <-> Byte 2/Output
//     Standard Outputs/Fix01.N101/Q @bit 24 <-> Byte 3/Output
//   SODG11_SSCC610_2403701_PLC/SODG11_SSCC610_2403701_PLC Instance <-> EtherCAT Master (EtherCAT)/IC01.T01 (EK1100)/IC01.T16 (EK1122)/Fix01.N11 (EP1008-0002)
//     Standard Inputs/Fix01.N11/I <-> Channel 1/Input
//     Standard Inputs/Fix01.N11/I @bit 1 <-> Channel 2/Input
//     Standard Inputs/Fix01.N11/I @bit 2 <-> Channel 3/Input
//     Standard Inputs/Fix01.N11/I @bit 3 <-> Channel 4/Input
//     Standard Inputs/Fix01.N11/I @bit 4 <-> Channel 5/Input
//     Standard Inputs/Fix01.N11/I @bit 5 <-> Channel 6/Input
//     Standard Inputs/Fix01.N11/I @bit 6 <-> Channel 7/Input
//     Standard Inputs/Fix01.N11/I @bit 7 <-> Channel 8/Input
//     Standard Inputs/Fix01.N11/InfoData/State <-> InfoData/State
//     Standard Inputs/Fix01.N11/Wc_State <-> WcState/WcState
//   SODG11_SSCC610_2403701_PLC/SODG11_SSCC610_2403701_PLC Instance <-> EtherCAT Master (EtherCAT)/IC01.T01 (EK1100)/IC01.T16 (EK1122)/Fix01.N12 (EP1008-0002)
//     Standard Inputs/Fix01.N12/I <-> Channel 1/Input
//     Standard Inputs/Fix01.N12/I @bit 1 <-> Channel 2/Input
//     Standard Inputs/Fix01.N12/I @bit 2 <-> Channel 3/Input
//     Standard Inputs/Fix01.N12/I @bit 3 <-> Channel 4/Input
//     Standard Inputs/Fix01.N12/I @bit 4 <-> Channel 5/Input
//     Standard Inputs/Fix01.N12/I @bit 5 <-> Channel 6/Input
//     Standard Inputs/Fix01.N12/I @bit 6 <-> Channel 7/Input
//     Standard Inputs/Fix01.N12/I @bit 7 <-> Channel 8/Input
//     Standard Inputs/Fix01.N12/InfoData/State <-> InfoData/State
//     Standard Inputs/Fix01.N12/Wc_State <-> WcState/WcState
//   SODG11_SSCC610_2403701_PLC/SODG11_SSCC610_2403701_PLC Instance <-> EtherCAT Master (EtherCAT)/IC01.T01 (EK1100)/IC01.T16 (EK1122)/Fix01.N13 (EP1008-0002)
//     Standard Inputs/Fix01.N13/I <-> Channel 1/Input
//     Standard Inputs/Fix01.N13/I @bit 1 <-> Channel 2/Input
//     Standard Inputs/Fix01.N13/I @bit 2 <-> Channel 3/Input
//     Standard Inputs/Fix01.N13/I @bit 3 <-> Channel 4/Input
//     Standard Inputs/Fix01.N13/I @bit 4 <-> Channel 5/Input
//     Standard Inputs/Fix01.N13/I @bit 5 <-> Channel 6/Input
//     Standard Inputs/Fix01.N13/I @bit 6 <-> Channel 7/Input
//     Standard Inputs/Fix01.N13/I @bit 7 <-> Channel 8/Input
//     Standard Inputs/Fix01.N13/InfoData/State <-> InfoData/State
//     Standard Inputs/Fix01.N13/Wc_State <-> WcState/WcState
//   SODG11_SSCC610_2403701_PLC/SODG11_SSCC610_2403701_PLC Instance <-> EtherCAT Master (EtherCAT)/IC01.T01 (EK1100)/IC01.T16 (EK1122)/Fix01.N14 (EP1008-0002)
//     Standard Inputs/Fix01.N14/I <-> Channel 1/Input
//     Standard Inputs/Fix01.N14/I @bit 1 <-> Channel 2/Input
//     Standard Inputs/Fix01.N14/I @bit 2 <-> Channel 3/Input
//     Standard Inputs/Fix01.N14/I @bit 3 <-> Channel 4/Input
//     Standard Inputs/Fix01.N14/I @bit 4 <-> Channel 5/Input
//     Standard Inputs/Fix01.N14/I @bit 5 <-> Channel 6/Input
//     Standard Inputs/Fix01.N14/I @bit 6 <-> Channel 7/Input
//     Standard Inputs/Fix01.N14/I @bit 7 <-> Channel 8/Input
//     Standard Inputs/Fix01.N14/InfoData/State <-> InfoData/State
//     Standard Inputs/Fix01.N14/Wc_State <-> WcState/WcState
//   SODG11_SSCC610_2403701_PLC/SODG11_SSCC610_2403701_PLC Instance <-> EtherCAT Master (EtherCAT)/IC01.T01 (EK1100)/IC01.T16 (EK1122)/Fix01.N15 (EP1008-0002)
//     Standard Inputs/Fix01.N15/I <-> Channel 1/Input
//     Standard Inputs/Fix01.N15/I @bit 1 <-> Channel 2/Input
//     Standard Inputs/Fix01.N15/I @bit 2 <-> Channel 3/Input
//     Standard Inputs/Fix01.N15/I @bit 3 <-> Channel 4/Input
//     Standard Inputs/Fix01.N15/I @bit 4 <-> Channel 5/Input
//     Standard Inputs/Fix01.N15/I @bit 5 <-> Channel 6/Input
//     Standard Inputs/Fix01.N15/I @bit 6 <-> Channel 7/Input
//     Standard Inputs/Fix01.N15/I @bit 7 <-> Channel 8/Input
//     Standard Inputs/Fix01.N15/InfoData/State <-> InfoData/State
//     Standard Inputs/Fix01.N15/Wc_State <-> WcState/WcState
//   SODG11_SSCC610_2403701_PLC/SODG11_SSCC610_2403701_PLC Instance <-> EtherCAT Master (EtherCAT)/IC01.T01 (EK1100)/IC01.T16 (EK1122)/Fix01.N16 (EP1008-0002)
//     Standard Inputs/Fix01.N16/I <-> Channel 1/Input
//     Standard Inputs/Fix01.N16/I @bit 1 <-> Channel 2/Input
//     Standard Inputs/Fix01.N16/I @bit 2 <-> Channel 3/Input
//     Standard Inputs/Fix01.N16/I @bit 3 <-> Channel 4/Input
//     Standard Inputs/Fix01.N16/I @bit 4 <-> Channel 5/Input
//     Standard Inputs/Fix01.N16/I @bit 5 <-> Channel 6/Input
//     Standard Inputs/Fix01.N16/I @bit 6 <-> Channel 7/Input
//     Standard Inputs/Fix01.N16/I @bit 7 <-> Channel 8/Input
//     Standard Inputs/Fix01.N16/InfoData/State <-> InfoData/State
//     Standard Inputs/Fix01.N16/Wc_State <-> WcState/WcState
//   SODG11_SSCC610_2403701_PLC/SODG11_SSCC610_2403701_PLC Instance <-> EtherCAT Master (EtherCAT)/IC01.T01 (EK1100)/IC01.T16 (EK1122)/Fix01.N17 (EP1008-0002)
//     Standard Inputs/Fix01.N17/I <-> Channel 1/Input
//     Standard Inputs/Fix01.N17/I @bit 1 <-> Channel 2/Input
//     Standard Inputs/Fix01.N17/I @bit 2 <-> Channel 3/Input
//     Standard Inputs/Fix01.N17/I @bit 3 <-> Channel 4/Input
//     Standard Inputs/Fix01.N17/I @bit 4 <-> Channel 5/Input
//     Standard Inputs/Fix01.N17/I @bit 5 <-> Channel 6/Input
//     Standard Inputs/Fix01.N17/I @bit 6 <-> Channel 7/Input
//     Standard Inputs/Fix01.N17/I @bit 7 <-> Channel 8/Input
//     Standard Inputs/Fix01.N17/InfoData/State <-> InfoData/State
//     Standard Inputs/Fix01.N17/Wc_State <-> WcState/WcState
//   SODG11_SSCC610_2403701_PLC/SODG11_SSCC610_2403701_PLC Instance <-> EtherCAT Master (EtherCAT)/IC01.T01 (EK1100)/IC01.T16 (EK1122)/Fix01.N18 (EP1008-0002)
//     Standard Inputs/Fix01.N18/I <-> Channel 1/Input
//     Standard Inputs/Fix01.N18/I @bit 1 <-> Channel 2/Input
//     Standard Inputs/Fix01.N18/I @bit 2 <-> Channel 3/Input
//     Standard Inputs/Fix01.N18/I @bit 3 <-> Channel 4/Input
//     Standard Inputs/Fix01.N18/I @bit 4 <-> Channel 5/Input
//     Standard Inputs/Fix01.N18/I @bit 5 <-> Channel 6/Input
//     Standard Inputs/Fix01.N18/I @bit 6 <-> Channel 7/Input
//     Standard Inputs/Fix01.N18/I @bit 7 <-> Channel 8/Input
//     Standard Inputs/Fix01.N18/InfoData/State <-> InfoData/State
//     Standard Inputs/Fix01.N18/Wc_State <-> WcState/WcState
//   SODG11_SSCC610_2403701_PLC/SODG11_SSCC610_2403701_PLC Instance <-> EtherCAT Master (EtherCAT)/IC01.T01 (EK1100)/IC01.T16 (EK1122)/Fix01.N19 (EP1008-0002)
//     Standard Inputs/Fix01.N19/I <-> Channel 1/Input
//     Standard Inputs/Fix01.N19/I @bit 1 <-> Channel 2/Input
//     Standard Inputs/Fix01.N19/I @bit 2 <-> Channel 3/Input
//     Standard Inputs/Fix01.N19/I @bit 3 <-> Channel 4/Input
//     Standard Inputs/Fix01.N19/I @bit 4 <-> Channel 5/Input
//     Standard Inputs/Fix01.N19/I @bit 5 <-> Channel 6/Input
//     Standard Inputs/Fix01.N19/I @bit 6 <-> Channel 7/Input
//     Standard Inputs/Fix01.N19/I @bit 7 <-> Channel 8/Input
//     Standard Inputs/Fix01.N19/InfoData/State <-> InfoData/State
//     Standard Inputs/Fix01.N19/Wc_State <-> WcState/WcState
//   SODG11_SSCC610_2403701_PLC/SODG11_SSCC610_2403701_PLC Instance <-> EtherCAT Master (EtherCAT)/IC01.T01 (EK1100)/IC01.T16 (EK1122)/Fix01.N20 (EP1008-0002)
//     Standard Inputs/Fix01.N20/I <-> Channel 1/Input
//     Standard Inputs/Fix01.N20/I @bit 1 <-> Channel 2/Input
//     Standard Inputs/Fix01.N20/I @bit 2 <-> Channel 3/Input
//     Standard Inputs/Fix01.N20/I @bit 3 <-> Channel 4/Input
//     Standard Inputs/Fix01.N20/I @bit 4 <-> Channel 5/Input
//     Standard Inputs/Fix01.N20/I @bit 5 <-> Channel 6/Input
//     Standard Inputs/Fix01.N20/I @bit 6 <-> Channel 7/Input
//     Standard Inputs/Fix01.N20/I @bit 7 <-> Channel 8/Input
//     Standard Inputs/Fix01.N20/InfoData/State <-> InfoData/State
//     Standard Inputs/Fix01.N20/Wc_State <-> WcState/WcState
//   SODG11_SSCC610_2403701_PLC/SODG11_SSCC610_2403701_PLC Instance <-> EtherCAT Master (EtherCAT)/IC01.T01 (EK1100)/IC01.T16 (EK1122)/Fix01.N21 (EP1008-0002)
//     Standard Inputs/Fix01.N21/I <-> Channel 1/Input
//     Standard Inputs/Fix01.N21/I @bit 1 <-> Channel 2/Input
//     Standard Inputs/Fix01.N21/I @bit 2 <-> Channel 3/Input
//     Standard Inputs/Fix01.N21/I @bit 3 <-> Channel 4/Input
//     Standard Inputs/Fix01.N21/I @bit 4 <-> Channel 5/Input
//     Standard Inputs/Fix01.N21/I @bit 5 <-> Channel 6/Input
//     Standard Inputs/Fix01.N21/I @bit 6 <-> Channel 7/Input
//     Standard Inputs/Fix01.N21/I @bit 7 <-> Channel 8/Input
//     Standard Inputs/Fix01.N21/InfoData/State <-> InfoData/State
//     Standard Inputs/Fix01.N21/Wc_State <-> WcState/WcState
//   SODG11_SSCC610_2403701_PLC/SODG11_SSCC610_2403701_PLC Instance <-> EtherCAT Master (EtherCAT)/IC01.T01 (EK1100)/IC01.T16 (EK1122)/Fix01.N22 (EP1008-0002)
